# B&R Automation Studio project MVP_ACOPOStrak
Automation Studio 4.7.4.67 SP; technology packages: mapp 5.9.1, mappCockpit 5.9.0, mappMotion 5.9.2, mappView 5.9.1

## Configuration ACOPOStrak

CPU 5PC900.TS17-00, AutomationRuntime C4.72, Build 4.1.2, Safety 0.0, Vc V4.53.0

### IoMap.iom - 5PC900_TS17_00/IoMap.iom
```iecst
VAR_CONFIG
	::Safety:moduleOK AT %IX."epl_icn".ModuleOk;
	::Safety:resetNeeded AT %IX."epl_icn".resetNeeded;
	::Safety:resetSafety AT %QX."epl_icn".resetCommand;
	::Safety:safetyStarted AT %IX."epl_icn".safetyStarted;
	::Safety:safetyOK AT %IX."epl_icn".safetyOK;
END_VAR
```

## Configuration Safety

### Task classes (Cpu.sw)
```
Cyclic#4:
  Safety <- Safety.prg
  PB1 <- PB1.prg
  PP1 <- PP1.prg
  PP2 <- PP2.prg
  PB2 <- PB2.prg
  PP3 <- PP3.prg
  PB3 <- PB3.prg
  PP4 <- PP4.prg
  PP5 <- PP5.prg
Binaries: arsvcreg, udbdef, TCData, arflatprv, arcoal, mvLoader, FWRules, mCoWebSc, ashwd, ashwac, User, sysconf, asfw, arconfig, Role, iomap, Config
Libraries: DataObj, AsXml, standard, runtime, FileIO, astime, mpbase, SfDomVis, asiodiag, asieccon, aruser, brsystem, SfDomDrv, sys_lib, MpSfDomMgr, asusb, astcp
```

- Safety project (password-protected, skipped)

## Configuration Simulation

### Task classes (Cpu.sw)
```
Cyclic#1:
  Safety <- Safety.prg
  Receip_Han <- SequenceHandler.prg
  PB1 <- PB1.prg
  PP1 <- PP1.prg
  PP2 <- PP2.prg
  PB2 <- PB2.prg
  PP3 <- PP3.prg
  PB3 <- PB3.prg
  PP4 <- PP4.prg
  PP5 <- PP5.prg
  Vis <- Vis.prg
  StartMovem <- StartMovement.prg
DataObjects: McAcpSys
Binaries: TCData, udbdef, mvLoader, mCoWebSc, arsvcreg, McAcpDrv, Config_5, Config_4, AlarmCore, AlarmHist, Settings, ashwac, arconfig, asfw, TraceConfi, User, ashwd, iomap, Role, sysconf, Config_1, Config_3, Config_2, McAcpSim, McProfGen
Libraries: McAxis, McBase, McAcpTrak, brsystem, AsSem, sys_lib, runtime, operator, astime, AsIecCon, CoTrace, AsZip, FileIO, MpAlarmX, MpBase, MpAxis, McAcpAx, AsBrStr, AsIODiag, arflatprv, arcoal, powerlnk, dataobj, standard, MpSfDomMgr, SfDomDrv, SfDomVis, aruser, asusb, astcp
```

### Hardware
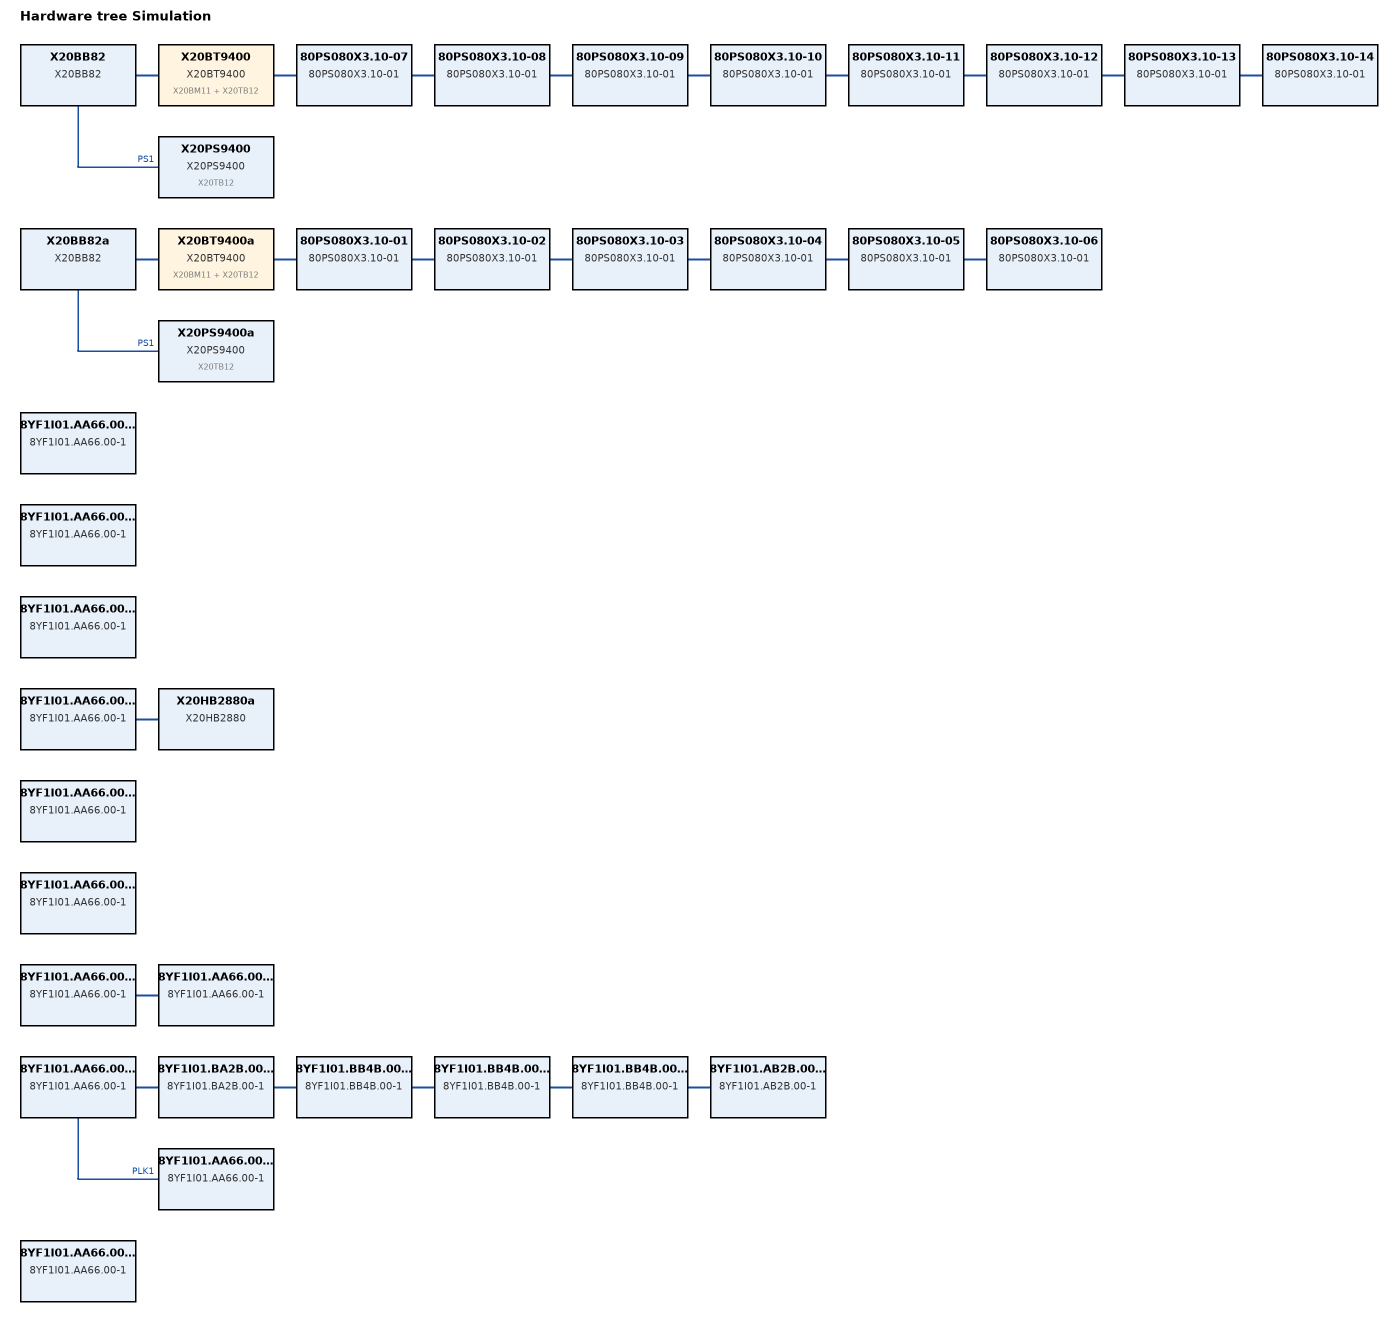
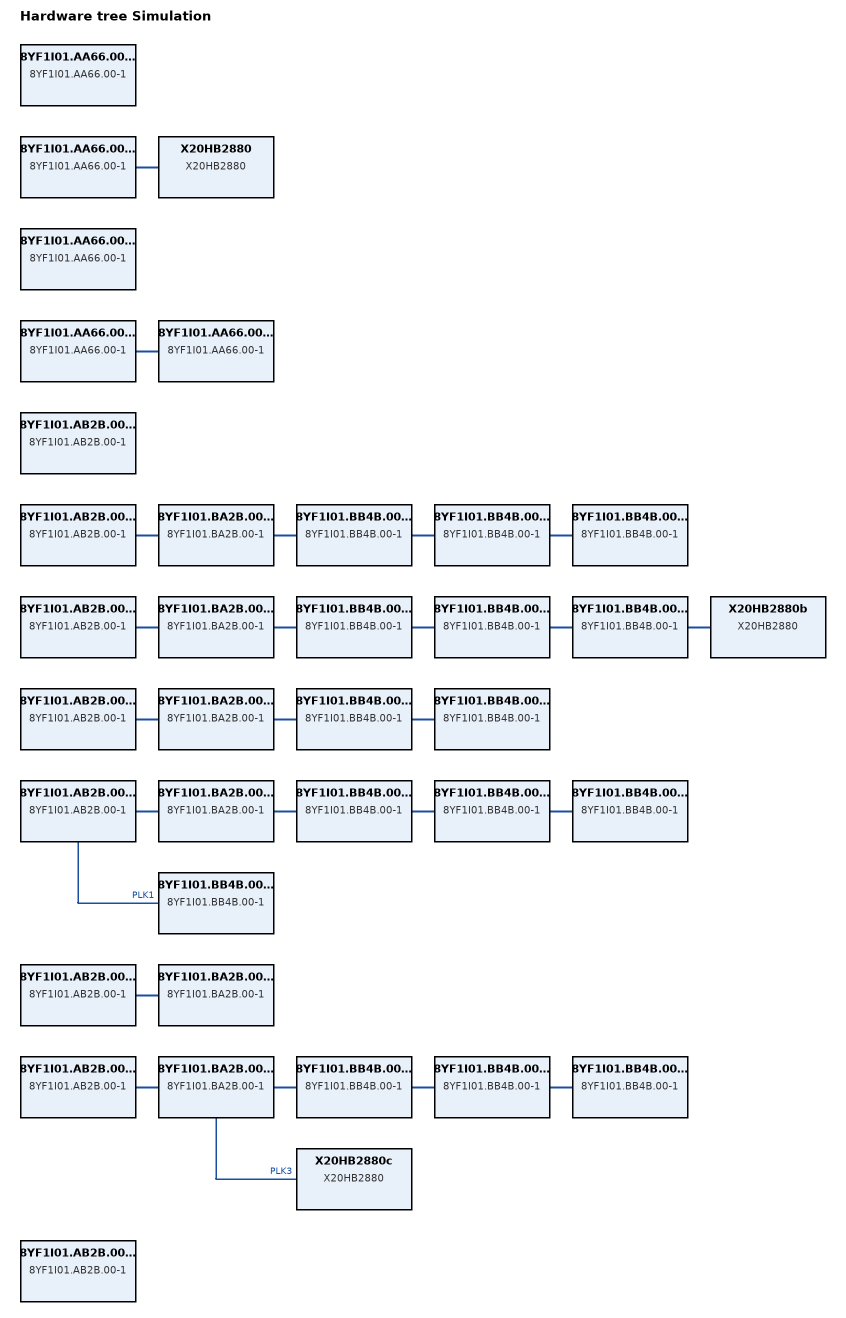
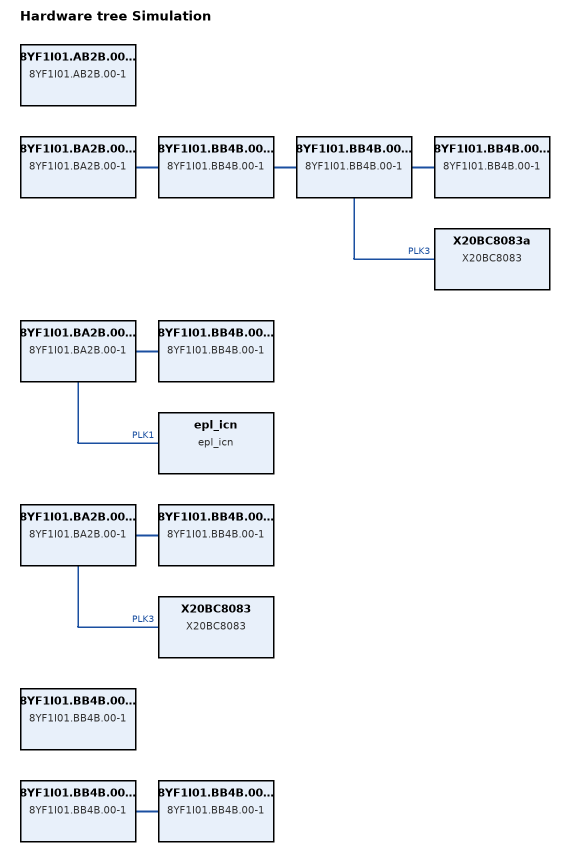
```
80PS080X3.10-01 : 80PS080X3.10-01 v1.3.0.0  [X2X1 -> X20BT9400a.X2X1 [Cable Type=X2XCable, Length=3, Version=1.0.0.2]]
  Supervision = off
  ParallelMode01 = on
  VoltageSet01 = 60
  ChopperEnable01 = on
80PS080X3.10-02 : 80PS080X3.10-01 v1.3.0.0  [X2X1 -> 80PS080X3.10-01.X2X2 [Cable Type=X2XCable, Length=1, Version=1.0.0.2]]
  Supervision = off
  ParallelMode01 = on
  VoltageSet01 = 60
  ChopperEnable01 = on
80PS080X3.10-03 : 80PS080X3.10-01 v1.3.0.0  [X2X1 -> 80PS080X3.10-02.X2X2 [Cable Type=X2XCable, Length=5, Version=1.0.0.2]]
  Supervision = off
  VoltageSet01 = 58
  ChopperEnable01 = on
80PS080X3.10-04 : 80PS080X3.10-01 v1.3.0.0  [X2X1 -> 80PS080X3.10-03.X2X2 [Cable Type=X2XCable, Length=1, Version=1.0.0.2]]
  Supervision = off
  VoltageSet01 = 58
  ChopperEnable01 = on
80PS080X3.10-05 : 80PS080X3.10-01 v1.3.0.0  [X2X1 -> 80PS080X3.10-04.X2X2 [Cable Type=X2XCable, Length=5, Version=1.0.0.2]]
  Supervision = off
  VoltageSet01 = 58
  ChopperEnable01 = on
80PS080X3.10-06 : 80PS080X3.10-01 v1.3.0.0  [X2X1 -> 80PS080X3.10-05.X2X2 [Cable Type=X2XCable, Length=1, Version=1.0.0.2]]
  Supervision = off
  VoltageSet01 = 58
  ChopperEnable01 = on
80PS080X3.10-07 : 80PS080X3.10-01 v1.3.0.0  [X2X1 -> X20BT9400.X2X1 [Cable Type=X2XCable, Length=5, Version=1.0.0.2]]
  Supervision = off
  VoltageSet01 = 58
  ChopperEnable01 = on
80PS080X3.10-08 : 80PS080X3.10-01 v1.3.0.0  [X2X1 -> 80PS080X3.10-07.X2X2 [Cable Type=X2XCable, Length=1, Version=1.0.0.2]]
  Supervision = off
  VoltageSet01 = 58
  ChopperEnable01 = on
80PS080X3.10-09 : 80PS080X3.10-01 v1.3.0.0  [X2X1 -> 80PS080X3.10-08.X2X2 [Cable Type=X2XCable, Length=1, Version=1.0.0.2]]
  Supervision = off
  VoltageSet01 = 58
  ChopperEnable01 = on
80PS080X3.10-10 : 80PS080X3.10-01 v1.3.0.0  [X2X1 -> 80PS080X3.10-09.X2X2 [Cable Type=X2XCable, Length=1, Version=1.0.0.2]]
  Supervision = off
  VoltageSet01 = 58
  ChopperEnable01 = on
80PS080X3.10-11 : 80PS080X3.10-01 v1.3.0.0  [X2X1 -> 80PS080X3.10-10.X2X2 [Cable Type=X2XCable, Length=3, Version=1.0.0.2]]
  Supervision = off
  VoltageSet01 = 58
  ChopperEnable01 = on
80PS080X3.10-12 : 80PS080X3.10-01 v1.3.0.0  [X2X1 -> 80PS080X3.10-11.X2X2 [Cable Type=X2XCable, Length=1, Version=1.0.0.2]]
  Supervision = off
  VoltageSet01 = 58
  ChopperEnable01 = on
80PS080X3.10-13 : 80PS080X3.10-01 v1.3.0.0  [X2X1 -> 80PS080X3.10-12.X2X2 [Cable Type=X2XCable, Length=1, Version=1.0.0.2]]
  Supervision = off
  VoltageSet01 = 58
  ChopperEnable01 = on
80PS080X3.10-14 : 80PS080X3.10-01 v1.3.0.0  [X2X1 -> 80PS080X3.10-13.X2X2 [Cable Type=X2XCable, Length=1, Version=1.0.0.2]]
  Supervision = off
  VoltageSet01 = 58
  ChopperEnable01 = on
8YF1I01.AA66.00-1_16 : 8YF1I01.AA66.00-1 v0.0.0.4  [PLK1 -> 8YF1I01.AA66.00-1_17.PLK2 (NodeNumber=16) [Cable Type=PowerlinkCable, Length=10, Version=1.0.0.2]]
  DriveConfiguration:
    McTypeID = LLMConfig
  DriveConfiguration/Segment:
    Shape = STRAIGHT660
    SegmentReference = SEG_1_16
    StopReaction = UseAssemblySetting
    SpeedFilter = UseAssemblySetting
8YF1I01.AA66.00-1_17 : 8YF1I01.AA66.00-1 v0.0.0.4  [PLK1 -> 8YF1I01.AA66.00-1_18.PLK2 (NodeNumber=17) [Cable Type=PowerlinkCable, Length=10, Version=1.0.0.2]; PLK2 -> 8YF1I01.AA66.00-1_16.PLK1 (NodeNumber=17) [Cable Type=PowerlinkCable, Length=10, Version=1.0.0.2]]
  DriveConfiguration:
    McTypeID = LLMConfig
  DriveConfiguration/Segment:
    Shape = STRAIGHT660
    SegmentReference = SEG_1_17
    StopReaction = UseAssemblySetting
    SpeedFilter = UseAssemblySetting
8YF1I01.AA66.00-1_18 : 8YF1I01.AA66.00-1 v0.0.0.4  [PLK1 -> 8YF1I01.AA66.00-1_19.PLK2 (NodeNumber=18) [Cable Type=PowerlinkCable, Length=10, Version=1.0.0.2]; PLK2 -> 8YF1I01.AA66.00-1_17.PLK1 (NodeNumber=18) [Cable Type=PowerlinkCable, Length=10, Version=1.0.0.2]]
  DriveConfiguration:
    McTypeID = LLMConfig
  DriveConfiguration/Segment:
    Shape = STRAIGHT660
    SegmentReference = SEG_1_18
    StopReaction = UseAssemblySetting
    SpeedFilter = UseAssemblySetting
8YF1I01.AA66.00-1_19 : 8YF1I01.AA66.00-1 v0.0.0.4  [PLK1 -> 8YF1I01.AA66.00-1_20.PLK2 (NodeNumber=19) [Cable Type=PowerlinkCable, Length=10, Version=1.0.0.2]; PLK2 -> 8YF1I01.AA66.00-1_18.PLK1 (NodeNumber=19) [Cable Type=PowerlinkCable, Length=10, Version=1.0.0.2]; PLK3 -> X20HB2880a.ETH1 (NodeNumber=19) [Cable Type=PowerlinkCable, Length=10, Version=1.0.0.2]]
  DriveConfiguration:
    McTypeID = LLMConfig
  DriveConfiguration/Segment:
    Shape = STRAIGHT660
    SegmentReference = SEG_1_19
    StopReaction = UseAssemblySetting
    SpeedFilter = UseAssemblySetting
8YF1I01.AA66.00-1_20 : 8YF1I01.AA66.00-1 v0.0.0.4  [PLK1 -> 8YF1I01.AA66.00-1_21.PLK2 (NodeNumber=20) [Cable Type=PowerlinkCable, Length=10, Version=1.0.0.2]; PLK2 -> 8YF1I01.AA66.00-1_19.PLK1 (NodeNumber=20) [Cable Type=PowerlinkCable, Length=10, Version=1.0.0.2]]
  DriveConfiguration:
    McTypeID = LLMConfig
  DriveConfiguration/Segment:
    Shape = STRAIGHT660
    SegmentReference = SEG_1_20
    StopReaction = UseAssemblySetting
    SpeedFilter = UseAssemblySetting
8YF1I01.AA66.00-1_21 : 8YF1I01.AA66.00-1 v0.0.0.4  [PLK1 -> 8YF1I01.AA66.00-1_22.PLK2 [Cable Type=PowerlinkCable, Length=10, Version=1.0.0.2]; PLK2 -> 8YF1I01.AA66.00-1_20.PLK1 [Cable Type=PowerlinkCable, Length=10, Version=1.0.0.2]]
  DriveConfiguration:
    McTypeID = LLMConfig
  DriveConfiguration/Segment:
    Shape = STRAIGHT660
    SegmentReference = SEG_1_21
    StopReaction = UseAssemblySetting
    SpeedFilter = UseAssemblySetting
8YF1I01.AA66.00-1_22 : 8YF1I01.AA66.00-1 v0.0.0.4  [PLK1 -> 8YF1I01.AA66.00-1_23.PLK2 [Cable Type=PowerlinkCable, Length=10, Version=1.0.0.2]; PLK2 -> 8YF1I01.AA66.00-1_21.PLK1 [Cable Type=PowerlinkCable, Length=10, Version=1.0.0.2]]
  DriveConfiguration:
    McTypeID = LLMConfig
  DriveConfiguration/Segment:
    Shape = STRAIGHT660
    SegmentReference = SEG_1_22
    StopReaction = UseAssemblySetting
    SpeedFilter = UseAssemblySetting
8YF1I01.AA66.00-1_23 : 8YF1I01.AA66.00-1 v0.0.0.4  [PLK2 -> 8YF1I01.AA66.00-1_22.PLK1 [Cable Type=PowerlinkCable, Length=10, Version=1.0.0.2]]
  DriveConfiguration:
    McTypeID = LLMConfig
  DriveConfiguration/Segment:
    Shape = STRAIGHT660
    SegmentReference = SEG_1_23
    StopReaction = UseAssemblySetting
    SpeedFilter = UseAssemblySetting
8YF1I01.AA66.00-1_29 : 8YF1I01.AA66.00-1 v0.0.0.4  [PLK1 -> 8YF1I01.AA66.00-1_30.PLK2 [Cable Type=PowerlinkCable, Length=10, Version=1.0.0.2]; PLK2 -> 8YF1I01.BA2B.00-1_28.PLK1 [Cable Type=PowerlinkCable, Length=10, Version=1.0.0.2]]
  DriveConfiguration:
    McTypeID = LLMConfig
  DriveConfiguration/Segment:
    Shape = STRAIGHT660
    SegmentReference = SEG_1_29
    StopReaction = UseAssemblySetting
    SpeedFilter = UseAssemblySetting
8YF1I01.AA66.00-1_30 : 8YF1I01.AA66.00-1 v0.0.0.4  [PLK2 -> 8YF1I01.AA66.00-1_29.PLK1 (NodeNumber=30) [Cable Type=PowerlinkCable, Length=10, Version=1.0.0.2]]
  DriveConfiguration:
    McTypeID = LLMConfig
  DriveConfiguration/Segment:
    Shape = STRAIGHT660
    SegmentReference = SEG_1_30
    StopReaction = UseAssemblySetting
    SpeedFilter = UseAssemblySetting
8YF1I01.AA66.00-1_31 : 8YF1I01.AA66.00-1 v0.0.0.4  [PLK1 -> 8YF1I01.AA66.00-1_32.PLK2 (NodeNumber=31) [Cable Type=PowerlinkCable, Length=10, Version=1.0.0.2]]
  DriveConfiguration:
    McTypeID = LLMConfig
  DriveConfiguration/Segment:
    Shape = STRAIGHT660
    SegmentReference = SEG_1_31
    StopReaction = UseAssemblySetting
    SpeedFilter = UseAssemblySetting
8YF1I01.AA66.00-1_32 : 8YF1I01.AA66.00-1 v0.0.0.4  [PLK1 -> 8YF1I01.AA66.00-1_33.PLK2 (NodeNumber=32) [Cable Type=PowerlinkCable, Length=10, Version=1.0.0.2]; PLK2 -> 8YF1I01.AA66.00-1_31.PLK1 (NodeNumber=32) [Cable Type=PowerlinkCable, Length=10, Version=1.0.0.2]]
  DriveConfiguration:
    McTypeID = LLMConfig
  DriveConfiguration/Segment:
    Shape = STRAIGHT660
    SegmentReference = SEG_1_32
    StopReaction = UseAssemblySetting
    SpeedFilter = UseAssemblySetting
8YF1I01.AA66.00-1_33 : 8YF1I01.AA66.00-1 v0.0.0.4  [PLK1 -> 8YF1I01.AA66.00-1_34.PLK2 (NodeNumber=33) [Cable Type=PowerlinkCable, Length=10, Version=1.0.0.2]; PLK2 -> 8YF1I01.AA66.00-1_32.PLK1 (NodeNumber=33) [Cable Type=PowerlinkCable, Length=10, Version=1.0.0.2]; PLK3 -> X20HB2880.ETH1 (NodeNumber=33) [Cable Type=PowerlinkCable, Length=10, Version=1.0.0.2]]
  DriveConfiguration:
    McTypeID = LLMConfig
  DriveConfiguration/Segment:
    Shape = STRAIGHT660
    SegmentReference = SEG_1_33
    StopReaction = UseAssemblySetting
    SpeedFilter = UseAssemblySetting
8YF1I01.AA66.00-1_34 : 8YF1I01.AA66.00-1 v0.0.0.4  [PLK1 -> 8YF1I01.AA66.00-1_35.PLK2 [Cable Type=PowerlinkCable, Length=10, Version=1.0.0.2]; PLK2 -> 8YF1I01.AA66.00-1_33.PLK1 [Cable Type=PowerlinkCable, Length=10, Version=1.0.0.2]]
  DriveConfiguration:
    McTypeID = LLMConfig
  DriveConfiguration/Segment:
    Shape = STRAIGHT660
    SegmentReference = SEG_1_34
    StopReaction = UseAssemblySetting
    SpeedFilter = UseAssemblySetting
8YF1I01.AA66.00-1_35 : 8YF1I01.AA66.00-1 v0.0.0.4  [PLK1 -> 8YF1I01.AA66.00-1_36.PLK2 [Cable Type=PowerlinkCable, Length=10, Version=1.0.0.2]; PLK2 -> 8YF1I01.AA66.00-1_34.PLK1 [Cable Type=PowerlinkCable, Length=10, Version=1.0.0.2]]
  DriveConfiguration:
    McTypeID = LLMConfig
  DriveConfiguration/Segment:
    Shape = STRAIGHT660
    SegmentReference = SEG_1_35
    StopReaction = UseAssemblySetting
    SpeedFilter = UseAssemblySetting
8YF1I01.AA66.00-1_36 : 8YF1I01.AA66.00-1 v0.0.0.4  [PLK2 -> 8YF1I01.AA66.00-1_35.PLK1 [Cable Type=PowerlinkCable, Length=10, Version=1.0.0.2]]
  DriveConfiguration:
    McTypeID = LLMConfig
  DriveConfiguration/Segment:
    Shape = STRAIGHT660
    SegmentReference = SEG_1_36
    StopReaction = UseAssemblySetting
    SpeedFilter = UseAssemblySetting
8YF1I01.AB2B.00-1_11 : 8YF1I01.AB2B.00-1 v0.0.0.4  [PLK1 -> 8YF1I01.BB4B.00-1_12.PLK2 (NodeNumber=11) [Cable Type=PowerlinkCable, Length=10, Version=1.0.0.2]]
  DriveConfiguration:
    McTypeID = LLMConfig
  DriveConfiguration/Segment:
    Shape = STRAIGHT105_TO_CIRCULAR
    SegmentReference = SEG_1_11
    StopReaction = UseAssemblySetting
    SpeedFilter = UseAssemblySetting
8YF1I01.AB2B.00-1_24 : 8YF1I01.AB2B.00-1 v0.0.0.4  [PLK1 -> 8YF1I01.BB4B.00-1_25.PLK2 (NodeNumber=24) [Cable Type=PowerlinkCable, Length=10, Version=1.0.0.2]]
  DriveConfiguration:
    McTypeID = LLMConfig
  DriveConfiguration/Segment:
    Shape = STRAIGHT105_TO_CIRCULAR
    SegmentReference = SEG_1_24
    StopReaction = UseAssemblySetting
    SpeedFilter = UseAssemblySetting
8YF1I01.AB2B.00-2_78 : 8YF1I01.AB2B.00-1 v0.0.0.4  [PLK1 -> 8YF1I01.BB4B.00-2_79.PLK2 (NodeNumber=78) [Cable Type=PowerlinkCable, Length=10, Version=1.0.0.2]; PLK2 -> 8YF1I01.BA2B.00-2_77.PLK1 (NodeNumber=78) [Cable Type=PowerlinkCable, Length=10, Version=1.0.0.2]]
  DriveConfiguration:
    McTypeID = LLMConfig
  DriveConfiguration/Segment:
    Shape = STRAIGHT105_TO_CIRCULAR
    SegmentReference = SEG_2_78
    StopReaction = UseAssemblySetting
    SpeedFilter = UseAssemblySetting
8YF1I01.AB2B.00-2_83 : 8YF1I01.AB2B.00-1 v0.0.0.4  [PLK2 -> 8YF1I01.BA2B.00-2_82.PLK1 [Cable Type=PowerlinkCable, Length=10, Version=1.0.0.2]]
  DriveConfiguration:
    McTypeID = LLMConfig
  DriveConfiguration/Segment:
    Shape = STRAIGHT105_TO_CIRCULAR
    SegmentReference = SEG_2_83
    StopReaction = UseAssemblySetting
    SpeedFilter = UseAssemblySetting
8YF1I01.AB2B.00-3_67 : 8YF1I01.AB2B.00-1 v0.0.0.4  [PLK1 -> 8YF1I01.BB4B.00-3_68.PLK2 (NodeNumber=67) [Cable Type=PowerlinkCable, Length=10, Version=1.0.0.2]; PLK2 -> 8YF1I01.BA2B.00-3_66.PLK1 (NodeNumber=67) [Cable Type=PowerlinkCable, Length=10, Version=1.0.0.2]]
  DriveConfiguration:
    McTypeID = LLMConfig
  DriveConfiguration/Segment:
    Shape = STRAIGHT105_TO_CIRCULAR
    SegmentReference = SEG_3_67
    StopReaction = UseAssemblySetting
    SpeedFilter = UseAssemblySetting
8YF1I01.AB2B.00-3_72 : 8YF1I01.AB2B.00-1 v0.0.0.4  [PLK1 -> 8YF1I01.BB4B.00-3_73.PLK2 [Cable Type=PowerlinkCable, Length=10, Version=1.0.0.2]; PLK2 -> 8YF1I01.BA2B.00-3_71.PLK1 [Cable Type=PowerlinkCable, Length=10, Version=1.0.0.2]]
  DriveConfiguration:
    McTypeID = LLMConfig
  DriveConfiguration/Segment:
    Shape = STRAIGHT105_TO_CIRCULAR
    SegmentReference = SEG_3_72
    StopReaction = UseAssemblySetting
    SpeedFilter = UseAssemblySetting
8YF1I01.AB2B.00-4_55 : 8YF1I01.AB2B.00-1 v0.0.0.4  [PLK1 -> 8YF1I01.BB4B.00-4_56.PLK2 (NodeNumber=55) [Cable Type=PowerlinkCable, Length=10, Version=1.0.0.2]; PLK2 -> 8YF1I01.BA2B.00-4_54.PLK1 (NodeNumber=55) [Cable Type=PowerlinkCable, Length=10, Version=1.0.0.2]]
  DriveConfiguration:
    McTypeID = LLMConfig
  DriveConfiguration/Segment:
    Shape = STRAIGHT105_TO_CIRCULAR
    SegmentReference = SEG_4_55
    StopReaction = UseAssemblySetting
    SpeedFilter = UseAssemblySetting
8YF1I01.AB2B.00-4_60 : 8YF1I01.AB2B.00-1 v0.0.0.4  [PLK1 -> 8YF1I01.BB4B.00-4_61.PLK2 [Cable Type=PowerlinkCable, Length=10, Version=1.0.0.2]; PLK2 -> 8YF1I01.BA2B.00-4_59.PLK1 [Cable Type=PowerlinkCable, Length=10, Version=1.0.0.2]]
  DriveConfiguration:
    McTypeID = LLMConfig
  DriveConfiguration/Segment:
    Shape = STRAIGHT105_TO_CIRCULAR
    SegmentReference = SEG_4_60
    StopReaction = UseAssemblySetting
    SpeedFilter = UseAssemblySetting
8YF1I01.AB2B.00-5_37 : 8YF1I01.AB2B.00-1 v0.0.0.4  [PLK1 -> 8YF1I01.BB4B.00-5_38.PLK2 (NodeNumber=37) [Cable Type=PowerlinkCable, Length=10, Version=1.0.0.2]; PLK3 -> X20HB2880.ETH2 (NodeNumber=37) [Cable Type=PowerlinkCable, Length=10, Version=1.0.0.2]]
  DriveConfiguration:
    McTypeID = LLMConfig
  DriveConfiguration/Segment:
    Shape = STRAIGHT105_TO_CIRCULAR
    SegmentReference = SEG_5_37
    StopReaction = UseAssemblySetting
    SpeedFilter = UseAssemblySetting
8YF1I01.AB2B.00-6_51 : 8YF1I01.AB2B.00-1 v0.0.0.4  [PLK1 -> 8YF1I01.BB4B.00-6_52.PLK2 (NodeNumber=51) [Cable Type=PowerlinkCable, Length=10, Version=1.0.0.2]]
  DriveConfiguration:
    McTypeID = LLMConfig
  DriveConfiguration/Segment:
    Shape = STRAIGHT105_TO_CIRCULAR
    SegmentReference = SEG_6_51
    StopReaction = UseAssemblySetting
    SpeedFilter = UseAssemblySetting
8YF1I01.BA2B.00-1_15 : 8YF1I01.BA2B.00-1 v0.0.0.4  [PLK2 -> 8YF1I01.BB4B.00-1_14.PLK1 [Cable Type=PowerlinkCable, Length=10, Version=1.0.0.2]]
  DriveConfiguration:
    McTypeID = LLMConfig
  DriveConfiguration/Segment:
    Shape = CIRCULAR_TO_STRAIGHT105
    SegmentReference = SEG_1_15
    StopReaction = UseAssemblySetting
    SpeedFilter = UseAssemblySetting
8YF1I01.BA2B.00-1_28 : 8YF1I01.BA2B.00-1 v0.0.0.4  [PLK1 -> 8YF1I01.AA66.00-1_29.PLK2 (NodeNumber=28) [Cable Type=PowerlinkCable, Length=10, Version=1.0.0.2]; PLK2 -> 8YF1I01.BB4B.00-1_27.PLK1 (NodeNumber=28) [Cable Type=PowerlinkCable, Length=10, Version=1.0.0.2]; PLK3 -> X20HB2880a.ETH2 (NodeNumber=28) [Cable Type=PowerlinkCable, Length=10, Version=1.0.0.2]]
  DriveConfiguration:
    McTypeID = LLMConfig
  DriveConfiguration/Segment:
    Shape = CIRCULAR_TO_STRAIGHT105
    SegmentReference = SEG_1_28
    StopReaction = UseAssemblySetting
    SpeedFilter = UseAssemblySetting
8YF1I01.BA2B.00-2_77 : 8YF1I01.BA2B.00-1 v0.0.0.4  [PLK1 -> 8YF1I01.AB2B.00-2_78.PLK2 (NodeNumber=77) [Cable Type=PowerlinkCable, Length=10, Version=1.0.0.2]; PLK2 -> 8YF1I01.BB4B.00-2_76.PLK1 (NodeNumber=77) [Cable Type=PowerlinkCable, Length=10, Version=1.0.0.2]]
  DriveConfiguration:
    McTypeID = LLMConfig
  DriveConfiguration/Segment:
    Shape = CIRCULAR_TO_STRAIGHT105
    SegmentReference = SEG_2_77
    StopReaction = UseAssemblySetting
    SpeedFilter = UseAssemblySetting
8YF1I01.BA2B.00-2_82 : 8YF1I01.BA2B.00-1 v0.0.0.4  [PLK1 -> 8YF1I01.AB2B.00-2_83.PLK2 [Cable Type=PowerlinkCable, Length=10, Version=1.0.0.2]; PLK2 -> 8YF1I01.BB4B.00-2_81.PLK1 [Cable Type=PowerlinkCable, Length=10, Version=1.0.0.2]]
  DriveConfiguration:
    McTypeID = LLMConfig
  DriveConfiguration/Segment:
    Shape = CIRCULAR_TO_STRAIGHT105
    SegmentReference = SEG_2_82
    StopReaction = UseAssemblySetting
    SpeedFilter = UseAssemblySetting
8YF1I01.BA2B.00-3_66 : 8YF1I01.BA2B.00-1 v0.0.0.4  [PLK1 -> 8YF1I01.AB2B.00-3_67.PLK2 (NodeNumber=66) [Cable Type=PowerlinkCable, Length=10, Version=1.0.0.2]; PLK2 -> 8YF1I01.BB4B.00-3_65.PLK1 (NodeNumber=66) [Cable Type=PowerlinkCable, Length=10, Version=1.0.0.2]]
  DriveConfiguration:
    McTypeID = LLMConfig
  DriveConfiguration/Segment:
    Shape = CIRCULAR_TO_STRAIGHT105
    SegmentReference = SEG_3_66
    StopReaction = UseAssemblySetting
    SpeedFilter = UseAssemblySetting
8YF1I01.BA2B.00-3_71 : 8YF1I01.BA2B.00-1 v0.0.0.4  [PLK1 -> 8YF1I01.AB2B.00-3_72.PLK2 [Cable Type=PowerlinkCable, Length=10, Version=1.0.0.2]; PLK2 -> 8YF1I01.BB4B.00-3_70.PLK1 [Cable Type=PowerlinkCable, Length=10, Version=1.0.0.2]]
  DriveConfiguration:
    McTypeID = LLMConfig
  DriveConfiguration/Segment:
    Shape = CIRCULAR_TO_STRAIGHT105
    SegmentReference = SEG_3_71
    StopReaction = UseAssemblySetting
    SpeedFilter = UseAssemblySetting
8YF1I01.BA2B.00-4_54 : 8YF1I01.BA2B.00-1 v0.0.0.4  [PLK1 -> 8YF1I01.AB2B.00-4_55.PLK2 (NodeNumber=54) [Cable Type=PowerlinkCable, Length=10, Version=1.0.0.2]]
  DriveConfiguration:
    McTypeID = LLMConfig
  DriveConfiguration/Segment:
    Shape = CIRCULAR_TO_STRAIGHT105
    SegmentReference = SEG_4_54
    StopReaction = UseAssemblySetting
    SpeedFilter = UseAssemblySetting
8YF1I01.BA2B.00-4_59 : 8YF1I01.BA2B.00-1 v0.0.0.4  [PLK1 -> 8YF1I01.AB2B.00-4_60.PLK2 (NodeNumber=59) [Cable Type=PowerlinkCable, Length=10, Version=1.0.0.2]; PLK2 -> 8YF1I01.BB4B.00-4_58.PLK1 (NodeNumber=59) [Cable Type=PowerlinkCable, Length=10, Version=1.0.0.2]; PLK3 -> X20HB2880c.ETH1 (NodeNumber=59) [Cable Type=PowerlinkCable, Length=10, Version=1.0.0.2]]
  DriveConfiguration:
    McTypeID = LLMConfig
  DriveConfiguration/Segment:
    Shape = CIRCULAR_TO_STRAIGHT105
    SegmentReference = SEG_4_59
    StopReaction = UseAssemblySetting
    SpeedFilter = UseAssemblySetting
8YF1I01.BA2B.00-5_39 : 8YF1I01.BA2B.00-1 v0.0.0.4  [PLK1 -> epl_icn.PLK1 [Cable Type=PowerlinkCable, Length=10, Version=1.0.0.2]; PLK2 -> 8YF1I01.BB4B.00-5_38.PLK1 [Cable Type=PowerlinkCable, Length=10, Version=1.0.0.2]]
  DriveConfiguration:
    McTypeID = LLMConfig
  DriveConfiguration/Segment:
    Shape = CIRCULAR_TO_STRAIGHT105
    SegmentReference = SEG_5_39
    StopReaction = UseAssemblySetting
    SpeedFilter = UseAssemblySetting
8YF1I01.BA2B.00-6_53 : 8YF1I01.BA2B.00-1 v0.0.0.4  [PLK2 -> 8YF1I01.BB4B.00-6_52.PLK1 (NodeNumber=53) [Cable Type=PowerlinkCable, Length=10, Version=1.0.0.2]; PLK3 -> X20BC8083.PLK2 (NodeNumber=53) [Cable Type=PowerlinkCable, Length=10, Version=1.0.0.2]]
  DriveConfiguration:
    McTypeID = LLMConfig
  DriveConfiguration/Segment:
    Shape = CIRCULAR_TO_STRAIGHT105
    SegmentReference = SEG_6_53
    StopReaction = UseAssemblySetting
    SpeedFilter = UseAssemblySetting
8YF1I01.BB4B.00-1_12 : 8YF1I01.BB4B.00-1 v0.0.0.4  [PLK1 -> 8YF1I01.BB4B.00-1_13.PLK2 (NodeNumber=12) [Cable Type=PowerlinkCable, Length=10, Version=1.0.0.2]; PLK2 -> 8YF1I01.AB2B.00-1_11.PLK1 (NodeNumber=12) [Cable Type=PowerlinkCable, Length=10, Version=1.0.0.2]]
  DriveConfiguration:
    McTypeID = LLMConfig
  DriveConfiguration/Segment:
    Shape = CIRCULAR
    SegmentReference = SEG_1_12
    StopReaction = UseAssemblySetting
    SpeedFilter = UseAssemblySetting
8YF1I01.BB4B.00-1_13 : 8YF1I01.BB4B.00-1 v0.0.0.4  [PLK1 -> 8YF1I01.BB4B.00-1_14.PLK2 (NodeNumber=13) [Cable Type=PowerlinkCable, Length=10, Version=1.0.0.2]; PLK2 -> 8YF1I01.BB4B.00-1_12.PLK1 (NodeNumber=13) [Cable Type=PowerlinkCable, Length=10, Version=1.0.0.2]; PLK3 -> X20BC8083a.PLK2 (NodeNumber=13) [Cable Type=PowerlinkCable, Length=10, Version=1.0.0.2]]
  DriveConfiguration:
    McTypeID = LLMConfig
  DriveConfiguration/Segment:
    Shape = CIRCULAR
    SegmentReference = SEG_1_13
    StopReaction = UseAssemblySetting
    SpeedFilter = UseAssemblySetting
8YF1I01.BB4B.00-1_14 : 8YF1I01.BB4B.00-1 v0.0.0.4  [PLK1 -> 8YF1I01.BA2B.00-1_15.PLK2 [Cable Type=PowerlinkCable, Length=10, Version=1.0.0.2]; PLK2 -> 8YF1I01.BB4B.00-1_13.PLK1 [Cable Type=PowerlinkCable, Length=10, Version=1.0.0.2]]
  DriveConfiguration:
    McTypeID = LLMConfig
  DriveConfiguration/Segment:
    Shape = CIRCULAR
    SegmentReference = SEG_1_14
    StopReaction = UseAssemblySetting
    SpeedFilter = UseAssemblySetting
8YF1I01.BB4B.00-1_25 : 8YF1I01.BB4B.00-1 v0.0.0.4  [PLK1 -> 8YF1I01.BB4B.00-1_26.PLK2 (NodeNumber=25) [Cable Type=PowerlinkCable, Length=10, Version=1.0.0.2]; PLK2 -> 8YF1I01.AB2B.00-1_24.PLK1 (NodeNumber=25) [Cable Type=PowerlinkCable, Length=10, Version=1.0.0.2]]
  DriveConfiguration:
    McTypeID = LLMConfig
  DriveConfiguration/Segment:
    Shape = CIRCULAR
    SegmentReference = SEG_1_25
    StopReaction = UseAssemblySetting
    SpeedFilter = UseAssemblySetting
8YF1I01.BB4B.00-1_26 : 8YF1I01.BB4B.00-1 v0.0.0.4  [PLK1 -> 8YF1I01.BB4B.00-1_27.PLK2 (NodeNumber=26) [Cable Type=PowerlinkCable, Length=10, Version=1.0.0.2]; PLK2 -> 8YF1I01.BB4B.00-1_25.PLK1 (NodeNumber=26) [Cable Type=PowerlinkCable, Length=10, Version=1.0.0.2]]
  DriveConfiguration:
    McTypeID = LLMConfig
  DriveConfiguration/Segment:
    Shape = CIRCULAR
    SegmentReference = SEG_1_26
    StopReaction = UseAssemblySetting
    SpeedFilter = UseAssemblySetting
8YF1I01.BB4B.00-1_27 : 8YF1I01.BB4B.00-1 v0.0.0.4  [PLK1 -> 8YF1I01.BA2B.00-1_28.PLK2 (NodeNumber=27) [Cable Type=PowerlinkCable, Length=10, Version=1.0.0.2]; PLK2 -> 8YF1I01.BB4B.00-1_26.PLK1 (NodeNumber=27) [Cable Type=PowerlinkCable, Length=10, Version=1.0.0.2]]
  DriveConfiguration:
    McTypeID = LLMConfig
  DriveConfiguration/Segment:
    Shape = CIRCULAR
    SegmentReference = SEG_1_27
    StopReaction = UseAssemblySetting
    SpeedFilter = UseAssemblySetting
8YF1I01.BB4B.00-2_74 : 8YF1I01.BB4B.00-1 v0.0.0.4  [PLK1 -> 8YF1I01.BB4B.00-2_75.PLK2 (NodeNumber=74) [Cable Type=PowerlinkCable, Length=10, Version=1.0.0.2]]
  DriveConfiguration:
    McTypeID = LLMConfig
  DriveConfiguration/Segment:
    Shape = CIRCULAR
    SegmentReference = SEG_2_74
    StopReaction = UseAssemblySetting
    SpeedFilter = UseAssemblySetting
8YF1I01.BB4B.00-2_75 : 8YF1I01.BB4B.00-1 v0.0.0.4  [PLK1 -> 8YF1I01.BB4B.00-2_76.PLK2 (NodeNumber=75) [Cable Type=PowerlinkCable, Length=10, Version=1.0.0.2]; PLK2 -> 8YF1I01.BB4B.00-2_74.PLK1 (NodeNumber=75) [Cable Type=PowerlinkCable, Length=10, Version=1.0.0.2]]
  DriveConfiguration:
    McTypeID = LLMConfig
  DriveConfiguration/Segment:
    Shape = CIRCULAR
    SegmentReference = SEG_2_75
    StopReaction = UseAssemblySetting
    SpeedFilter = UseAssemblySetting
8YF1I01.BB4B.00-2_76 : 8YF1I01.BB4B.00-1 v0.0.0.4  [PLK1 -> 8YF1I01.BA2B.00-2_77.PLK2 (NodeNumber=76) [Cable Type=PowerlinkCable, Length=10, Version=1.0.0.2]; PLK2 -> 8YF1I01.BB4B.00-2_75.PLK1 (NodeNumber=76) [Cable Type=PowerlinkCable, Length=10, Version=1.0.0.2]]
  DriveConfiguration:
    McTypeID = LLMConfig
  DriveConfiguration/Segment:
    Shape = CIRCULAR
    SegmentReference = SEG_2_76
    StopReaction = UseAssemblySetting
    SpeedFilter = UseAssemblySetting
8YF1I01.BB4B.00-2_79 : 8YF1I01.BB4B.00-1 v0.0.0.4  [PLK1 -> 8YF1I01.BB4B.00-2_80.PLK2 (NodeNumber=79) [Cable Type=PowerlinkCable, Length=10, Version=1.0.0.2]; PLK2 -> 8YF1I01.AB2B.00-2_78.PLK1 (NodeNumber=79) [Cable Type=PowerlinkCable, Length=10, Version=1.0.0.2]; PLK3 -> X20HB2880b.ETH1 (NodeNumber=79) [Cable Type=PowerlinkCable, Length=10, Version=1.0.0.2]]
  DriveConfiguration:
    McTypeID = LLMConfig
  DriveConfiguration/Segment:
    Shape = CIRCULAR
    SegmentReference = SEG_2_79
    StopReaction = UseAssemblySetting
    SpeedFilter = UseAssemblySetting
8YF1I01.BB4B.00-2_80 : 8YF1I01.BB4B.00-1 v0.0.0.4  [PLK1 -> 8YF1I01.BB4B.00-2_81.PLK2 [Cable Type=PowerlinkCable, Length=10, Version=1.0.0.2]; PLK2 -> 8YF1I01.BB4B.00-2_79.PLK1 [Cable Type=PowerlinkCable, Length=10, Version=1.0.0.2]]
  DriveConfiguration:
    McTypeID = LLMConfig
  DriveConfiguration/Segment:
    Shape = CIRCULAR
    SegmentReference = SEG_2_80
    StopReaction = UseAssemblySetting
    SpeedFilter = UseAssemblySetting
8YF1I01.BB4B.00-2_81 : 8YF1I01.BB4B.00-1 v0.0.0.4  [PLK1 -> 8YF1I01.BA2B.00-2_82.PLK2 [Cable Type=PowerlinkCable, Length=10, Version=1.0.0.2]; PLK2 -> 8YF1I01.BB4B.00-2_80.PLK1 [Cable Type=PowerlinkCable, Length=10, Version=1.0.0.2]]
  DriveConfiguration:
    McTypeID = LLMConfig
  DriveConfiguration/Segment:
    Shape = CIRCULAR
    SegmentReference = SEG_2_81
    StopReaction = UseAssemblySetting
    SpeedFilter = UseAssemblySetting
8YF1I01.BB4B.00-3_64 : 8YF1I01.BB4B.00-1 v0.0.0.4  [PLK1 -> 8YF1I01.BB4B.00-3_65.PLK2 (NodeNumber=64) [Cable Type=PowerlinkCable, Length=10, Version=1.0.0.2]]
  DriveConfiguration:
    McTypeID = LLMConfig
  DriveConfiguration/Segment:
    Shape = CIRCULAR
    SegmentReference = SEG_3_64
    StopReaction = UseAssemblySetting
    SpeedFilter = UseAssemblySetting
8YF1I01.BB4B.00-3_65 : 8YF1I01.BB4B.00-1 v0.0.0.4  [PLK1 -> 8YF1I01.BA2B.00-3_66.PLK2 (NodeNumber=65) [Cable Type=PowerlinkCable, Length=10, Version=1.0.0.2]; PLK2 -> 8YF1I01.BB4B.00-3_64.PLK1 (NodeNumber=65) [Cable Type=PowerlinkCable, Length=10, Version=1.0.0.2]]
  DriveConfiguration:
    McTypeID = LLMConfig
  DriveConfiguration/Segment:
    Shape = CIRCULAR
    SegmentReference = SEG_3_65
    StopReaction = UseAssemblySetting
    SpeedFilter = UseAssemblySetting
8YF1I01.BB4B.00-3_68 : 8YF1I01.BB4B.00-1 v0.0.0.4  [PLK1 -> 8YF1I01.BB4B.00-3_69.PLK2 (NodeNumber=68) [Cable Type=PowerlinkCable, Length=10, Version=1.0.0.2]; PLK2 -> 8YF1I01.AB2B.00-3_67.PLK1 (NodeNumber=68) [Cable Type=PowerlinkCable, Length=10, Version=1.0.0.2]]
  DriveConfiguration:
    McTypeID = LLMConfig
  DriveConfiguration/Segment:
    Shape = CIRCULAR
    SegmentReference = SEG_3_68
    StopReaction = UseAssemblySetting
    SpeedFilter = UseAssemblySetting
8YF1I01.BB4B.00-3_69 : 8YF1I01.BB4B.00-1 v0.0.0.4  [PLK1 -> 8YF1I01.BB4B.00-3_70.PLK2 (NodeNumber=69) [Cable Type=PowerlinkCable, Length=10, Version=1.0.0.2]; PLK2 -> 8YF1I01.BB4B.00-3_68.PLK1 (NodeNumber=69) [Cable Type=PowerlinkCable, Length=10, Version=1.0.0.2]; PLK3 -> X20HB2880c.ETH2 (NodeNumber=69) [Cable Type=PowerlinkCable, Length=10, Version=1.0.0.2]]
  DriveConfiguration:
    McTypeID = LLMConfig
  DriveConfiguration/Segment:
    Shape = CIRCULAR
    SegmentReference = SEG_3_69
    StopReaction = UseAssemblySetting
    SpeedFilter = UseAssemblySetting
8YF1I01.BB4B.00-3_70 : 8YF1I01.BB4B.00-1 v0.0.0.4  [PLK1 -> 8YF1I01.BA2B.00-3_71.PLK2 [Cable Type=PowerlinkCable, Length=10, Version=1.0.0.2]; PLK2 -> 8YF1I01.BB4B.00-3_69.PLK1 [Cable Type=PowerlinkCable, Length=10, Version=1.0.0.2]]
  DriveConfiguration:
    McTypeID = LLMConfig
  DriveConfiguration/Segment:
    Shape = CIRCULAR
    SegmentReference = SEG_3_70
    StopReaction = UseAssemblySetting
    SpeedFilter = UseAssemblySetting
8YF1I01.BB4B.00-3_73 : 8YF1I01.BB4B.00-1 v0.0.0.4  [PLK2 -> 8YF1I01.AB2B.00-3_72.PLK1 [Cable Type=PowerlinkCable, Length=10, Version=1.0.0.2]]
  DriveConfiguration:
    McTypeID = LLMConfig
  DriveConfiguration/Segment:
    Shape = CIRCULAR
    SegmentReference = SEG_3_73
    StopReaction = UseAssemblySetting
    SpeedFilter = UseAssemblySetting
8YF1I01.BB4B.00-4_56 : 8YF1I01.BB4B.00-1 v0.0.0.4  [PLK1 -> 8YF1I01.BB4B.00-4_57.PLK2 (NodeNumber=56) [Cable Type=PowerlinkCable, Length=10, Version=1.0.0.2]; PLK2 -> 8YF1I01.AB2B.00-4_55.PLK1 (NodeNumber=56) [Cable Type=PowerlinkCable, Length=10, Version=1.0.0.2]]
  DriveConfiguration:
    McTypeID = LLMConfig
  DriveConfiguration/Segment:
    Shape = CIRCULAR
    SegmentReference = SEG_4_56
    StopReaction = UseAssemblySetting
    SpeedFilter = UseAssemblySetting
8YF1I01.BB4B.00-4_57 : 8YF1I01.BB4B.00-1 v0.0.0.4  [PLK1 -> 8YF1I01.BB4B.00-4_58.PLK2 (NodeNumber=57) [Cable Type=PowerlinkCable, Length=10, Version=1.0.0.2]; PLK2 -> 8YF1I01.BB4B.00-4_56.PLK1 (NodeNumber=57) [Cable Type=PowerlinkCable, Length=10, Version=1.0.0.2]]
  DriveConfiguration:
    McTypeID = LLMConfig
  DriveConfiguration/Segment:
    Shape = CIRCULAR
    SegmentReference = SEG_4_57
    StopReaction = UseAssemblySetting
    SpeedFilter = UseAssemblySetting
8YF1I01.BB4B.00-4_58 : 8YF1I01.BB4B.00-1 v0.0.0.4  [PLK1 -> 8YF1I01.BA2B.00-4_59.PLK2 (NodeNumber=58) [Cable Type=PowerlinkCable, Length=10, Version=1.0.0.2]; PLK2 -> 8YF1I01.BB4B.00-4_57.PLK1 (NodeNumber=58) [Cable Type=PowerlinkCable, Length=10, Version=1.0.0.2]]
  DriveConfiguration:
    McTypeID = LLMConfig
  DriveConfiguration/Segment:
    Shape = CIRCULAR
    SegmentReference = SEG_4_58
    StopReaction = UseAssemblySetting
    SpeedFilter = UseAssemblySetting
8YF1I01.BB4B.00-4_61 : 8YF1I01.BB4B.00-1 v0.0.0.4  [PLK1 -> 8YF1I01.BB4B.00-4_62.PLK2 [Cable Type=PowerlinkCable, Length=10, Version=1.0.0.2]; PLK2 -> 8YF1I01.AB2B.00-4_60.PLK1 [Cable Type=PowerlinkCable, Length=10, Version=1.0.0.2]]
  DriveConfiguration:
    McTypeID = LLMConfig
  DriveConfiguration/Segment:
    Shape = CIRCULAR
    SegmentReference = SEG_4_61
    StopReaction = UseAssemblySetting
    SpeedFilter = UseAssemblySetting
8YF1I01.BB4B.00-4_62 : 8YF1I01.BB4B.00-1 v0.0.0.4  [PLK1 -> 8YF1I01.BB4B.00-4_63.PLK2 (NodeNumber=62) [Cable Type=PowerlinkCable, Length=10, Version=1.0.0.2]; PLK2 -> 8YF1I01.BB4B.00-4_61.PLK1 (NodeNumber=62) [Cable Type=PowerlinkCable, Length=10, Version=1.0.0.2]]
  DriveConfiguration:
    McTypeID = LLMConfig
  DriveConfiguration/Segment:
    Shape = CIRCULAR
    SegmentReference = SEG_4_62
    StopReaction = UseAssemblySetting
    SpeedFilter = UseAssemblySetting
8YF1I01.BB4B.00-4_63 : 8YF1I01.BB4B.00-1 v0.0.0.4  [PLK2 -> 8YF1I01.BB4B.00-4_62.PLK1 [Cable Type=PowerlinkCable, Length=10, Version=1.0.0.2]]
  DriveConfiguration:
    McTypeID = LLMConfig
  DriveConfiguration/Segment:
    Shape = CIRCULAR
    SegmentReference = SEG_4_63
    StopReaction = UseAssemblySetting
    SpeedFilter = UseAssemblySetting
8YF1I01.BB4B.00-5_38 : 8YF1I01.BB4B.00-1 v0.0.0.4  [PLK1 -> 8YF1I01.BA2B.00-5_39.PLK2 [Cable Type=PowerlinkCable, Length=10, Version=1.0.0.2]; PLK2 -> 8YF1I01.AB2B.00-5_37.PLK1 [Cable Type=PowerlinkCable, Length=10, Version=1.0.0.2]]
  DriveConfiguration:
    McTypeID = LLMConfig
  DriveConfiguration/Segment:
    Shape = CIRCULAR
    SegmentReference = SEG_5_38
    StopReaction = UseAssemblySetting
    SpeedFilter = UseAssemblySetting
8YF1I01.BB4B.00-6_52 : 8YF1I01.BB4B.00-1 v0.0.0.4  [PLK1 -> 8YF1I01.BA2B.00-6_53.PLK2 (NodeNumber=52) [Cable Type=PowerlinkCable, Length=10, Version=1.0.0.2]; PLK2 -> 8YF1I01.AB2B.00-6_51.PLK1 (NodeNumber=52) [Cable Type=PowerlinkCable, Length=10, Version=1.0.0.2]]
  DriveConfiguration:
    McTypeID = LLMConfig
  DriveConfiguration/Segment:
    Shape = CIRCULAR
    SegmentReference = SEG_6_52
    StopReaction = UseAssemblySetting
    SpeedFilter = UseAssemblySetting
X20BB82 : X20BB82 v1.0.2.0
  Connector IF1:
    CycleTime = 10000
    BusLength = 50
    Stations = 32
    AsyncPayload = 96
X20BB82a : X20BB82 v1.0.2.0
  Connector IF1:
    CycleTime = 10000
    BusLength = 50
    Stations = 32
    AsyncPayload = 96
X20BC8083 : X20BC8083 v2.10.0.0  [PLK1 -> 5LS182.6-2.IF1 (NodeNumber=50) [Cable Type=PowerlinkCable, Length=10, Version=1.0.0.2]; PLK2 -> 8YF1I01.BA2B.00-6_53.PLK3 (NodeNumber=50) [Cable Type=PowerlinkCable, Length=10, Version=1.0.0.2]; SL -> X20BB82.SL1]
  Supervision = off
X20BC8083a : X20BC8083 v2.10.0.0  [PLK1 -> 5LS182.6-2.PLK2 (NodeNumber=10) [Cable Type=PowerlinkCable, Length=10, Version=1.0.0.2]; PLK2 -> 8YF1I01.BB4B.00-1_13.PLK3 (NodeNumber=10) [Cable Type=PowerlinkCable, Length=10, Version=1.0.0.2]; SL -> X20BB82a.SL1]
  Supervision = off
X20BM11 : X20BM11 v1.0.0.1  [X2X1 -> X20BB82.IF1]
X20BM11a : X20BM11 v1.0.0.1  [X2X1 -> X20BB82a.IF1]
X20BT9400 : X20BT9400 v1.1.0.0  [SS1 -> X20TB12b.SS; SL -> X20BM11.SL1]
  Supervision = off
  PowerInfo = on
X20BT9400a : X20BT9400 v1.1.0.0  [SS1 -> X20TB12c.SS; SL -> X20BM11a.SL1]
  Supervision = off
  PowerInfo = on
X20HB2880 : X20HB2880 v1.1.0.0  [ETH1 -> 8YF1I01.AA66.00-1_33.PLK3 [Cable Type=PowerlinkCable, Length=10, Version=1.0.0.2]; ETH2 -> 8YF1I01.AB2B.00-5_37.PLK3 [Cable Type=PowerlinkCable, Length=10, Version=1.0.0.2]; SS -> X20BB82a.SS2]
X20HB2880a : X20HB2880 v1.1.0.0  [ETH1 -> 8YF1I01.AA66.00-1_19.PLK3 [Cable Type=PowerlinkCable, Length=10, Version=1.0.0.2]; ETH2 -> 8YF1I01.BA2B.00-1_28.PLK3 [Cable Type=PowerlinkCable, Length=10, Version=1.0.0.2]; SS -> X20BB82a.SS1]
X20HB2880b : X20HB2880 v1.1.0.0  [ETH1 -> 8YF1I01.BB4B.00-2_79.PLK3 [Cable Type=PowerlinkCable, Length=10, Version=1.0.0.2]; SS -> X20BB82.SS2]
X20HB2880c : X20HB2880 v1.1.0.0  [ETH1 -> 8YF1I01.BA2B.00-4_59.PLK3 [Cable Type=PowerlinkCable, Length=10, Version=1.0.0.2]; ETH2 -> 8YF1I01.BB4B.00-3_69.PLK3 [Cable Type=PowerlinkCable, Length=10, Version=1.0.0.2]; SS -> X20BB82.SS1]
X20PS9400 : X20PS9400 v1.3.0.0  [SS1 -> X20TB12.SS; PS -> X20BB82.PS1]
  Supervision = off
  PowerInfo = on
X20PS9400a : X20PS9400 v1.3.0.0  [SS1 -> X20TB12a.SS; PS -> X20BB82a.PS1]
  Supervision = off
  PowerInfo = on
X20TB12 : X20TB12 v1.0.0.0
X20TB12a : X20TB12 v1.0.0.0
X20TB12b : X20TB12 v1.0.0.0
X20TB12c : X20TB12 v1.0.0.0
epl_icn : epl_icn v1.3.2.0  [PLK1 -> 8YF1I01.BA2B.00-5_39.PLK1 (NodeNumber=200) [Cable Type=PowerlinkCable, Length=10, Version=1.0.0.2]]
  RefConfiguration = Safety
  RefInterface = X20CP0484.IF3
```

### Config_1.assembly - 5PC900_TS17_00/mappMotion/Config_1.assembly
```
Element gAssembly_1 (Type=assembly)
  Tracks:
    TrackSeparation = 0.030
    Track[1]:
      Segments:
        SegmentRef[1] = ::SEG_1_11
        SegmentRef[2] = ::SEG_1_12
        SegmentRef[3] = ::SEG_1_13
        SegmentRef[4] = ::SEG_1_14
        SegmentRef[5] = ::SEG_1_15
        SegmentRef[6] = ::SEG_1_16
        SegmentRef[7] = ::SEG_1_17
        SegmentRef[8] = ::SEG_1_18
        SegmentRef[9] = ::SEG_1_19
        SegmentRef[10] = ::SEG_1_20
        SegmentRef[11] = ::SEG_1_21
        SegmentRef[12] = ::SEG_1_22
        SegmentRef[13] = ::SEG_1_23
        SegmentRef[14] = ::SEG_1_24
        SegmentRef[15] = ::SEG_1_25
        SegmentRef[16] = ::SEG_1_26
        SegmentRef[17] = ::SEG_1_27
        SegmentRef[18] = ::SEG_1_28
        SegmentRef[19] = ::SEG_1_29
        SegmentRef[20] = ::SEG_1_30
        SegmentRef[21] = ::SEG_1_31
        SegmentRef[22] = ::SEG_1_32
        SegmentRef[23] = ::SEG_1_33
        SegmentRef[24] = ::SEG_1_34
        SegmentRef[25] = ::SEG_1_35
        SegmentRef[26] = ::SEG_1_36
      Position = Absolute
        SegmentRef = ::SEG_1_21
        SegmentCountDirection = RightToLeft
        Translation:
          X = 0.0
          Y = 0.0
          Z = 0.0
        Orientation:
          Angle1 = 0.0
          Angle2 = 0.0
          Angle3 = 0
    Track[2]:
      Segments:
        SegmentRef[1] = ::SEG_2_74
        SegmentRef[2] = ::SEG_2_75
        SegmentRef[3] = ::SEG_2_76
        SegmentRef[4] = ::SEG_2_77
        SegmentRef[5] = ::SEG_2_78
        SegmentRef[6] = ::SEG_2_79
        SegmentRef[7] = ::SEG_2_80
        SegmentRef[8] = ::SEG_2_81
        SegmentRef[9] = ::SEG_2_82
        SegmentRef[10] = ::SEG_2_83
      Position = RelativeToOne
        TrackSegmentPosition:
          SegmentRef = ::SEG_2_77
          PositionRelativeTo = FromEnd
        Base:
          SegmentRef = ::SEG_1_29
          Position = 0.321
    Track[3]:
      Segments:
        SegmentRef[1] = ::SEG_3_64
        SegmentRef[2] = ::SEG_3_65
        SegmentRef[3] = ::SEG_3_66
        SegmentRef[4] = ::SEG_3_67
        SegmentRef[5] = ::SEG_3_68
        SegmentRef[6] = ::SEG_3_69
        SegmentRef[7] = ::SEG_3_70
        SegmentRef[8] = ::SEG_3_71
        SegmentRef[9] = ::SEG_3_72
        SegmentRef[10] = ::SEG_3_73
      Position = RelativeToOne
        TrackSegmentPosition:
          SegmentRef = ::SEG_3_66
          PositionRelativeTo = FromEnd
        Base:
          SegmentRef = ::SEG_1_34
          Position = 0.33
    Track[4]:
      Segments:
        SegmentRef[1] = ::SEG_4_54
        SegmentRef[2] = ::SEG_4_55
        SegmentRef[3] = ::SEG_4_56
        SegmentRef[4] = ::SEG_4_57
        SegmentRef[5] = ::SEG_4_58
        SegmentRef[6] = ::SEG_4_59
        SegmentRef[7] = ::SEG_4_60
        SegmentRef[8] = ::SEG_4_61
        SegmentRef[9] = ::SEG_4_62
        SegmentRef[10] = ::SEG_4_63
      Position = RelativeToOne
        TrackSegmentPosition:
          SegmentRef = ::SEG_4_59
          PositionRelativeTo = FromEnd
        Base:
          SegmentRef = ::SEG_1_19
          Position = 0.33
    Track[5]:
      Segments:
        SegmentRef[1] = ::SEG_5_37
        SegmentRef[2] = ::SEG_5_38
        SegmentRef[3] = ::SEG_5_39
      Position = RelativeToOne
        TrackSegmentPosition:
          SegmentRef = ::SEG_5_39
          PositionRelativeTo = FromEnd
        Base:
          SegmentRef = ::SEG_1_11
    Track[6]:
      Segments:
        SegmentRef[1] = ::SEG_6_51
        SegmentRef[2] = ::SEG_6_52
        SegmentRef[3] = ::SEG_6_53
      Position = RelativeToOne
        TrackSegmentPosition:
          SegmentRef = ::SEG_6_51
        Base:
          SegmentRef = ::SEG_1_15
          PositionRelativeTo = FromEnd
  CommonSegmentSettings:
    SegmentSimulationOnPLC = Off
    StopReaction = InductionHalt
    SpeedFilter = Lowpass
      FilterTime = 0.0004
    ControllerParameters:
      DefaultParameter:
        Controller:
          Position:
            ProportionalGain = 150.0
          Speed:
            ProportionalGain = 80.0
            IntegrationTime = 0.0
          FeedForward:
            TotalMass = 0.0
            ForcePositive = 0.0
            ForceNegative = 0.0
            SpeedForceFactor = 0.0
            ForceLoad = 0.0
        MovementErrorLimits:
          PositionError = 1.0
          VelocityError = 10.0
      AdditionalParameterSets = NotUsed
  Shuttles:
    MaxShuttleCount = 40
    ShuttleStereotypes:
      ShuttleStRef[1] = ShuttleStereotype_1
    MagnetPlateConfigurations:
      ShuttleType[1] = 8F1SA.100.xxxxxx-x
    CollisionAvoidance:
      Strategy = Constant
      MaximumModelDimensions:
        Length:
          ExtentToFront = 0.065
          ExtentToBack = 0.065
        Width:
          Width = 0.240
  AssemblyFeatures:
    AssemblyFeatureRef[1] = AssemblyFeature_2
  Visualization:
    MonitoringPv = ::gShuttleMon
    ProcessingTaskClass = 1
```

### Config_2.shuttlestereotype - 5PC900_TS17_00/mappMotion/Config_2.shuttlestereotype
```
Element ShuttleStereotype_1 (Type=shuttlestereotype)
  MeasurementUnit = 5067858
  MeasurementResolution = 0.00001
  MovementLimits = Internal
    VelocityIsReadOnly = 0
    Velocity:
      Velocity = 5
    AccelerationIsReadOnly = 0
    Acceleration:
      Acceleration = 50
    DecelerationIsReadOnly = 0
    Deceleration:
      Deceleration = 50
  JerkFilter = Used
    JerkTime = 0.02
  UserData:
    Size = 12
  CollisionAvoidance:
    InitialModelDimensions = UseExplicitValues
      Length:
        ExtentToFront = 0.040
        ExtentToBack = 0.040
      Width:
        Width = 0.080
```

### Config_3.sector - 5PC900_TS17_00/mappMotion/Config_3.sector
```
Element SectorTrack1 (Type=sector)
  Type = Composed
    StartSegment:
      SegmentRef = ::SEG_1_11
    IntermediateSegments:
      SegmentRef[1] = ::SEG_1_12
      SegmentRef[2] = ::SEG_1_13
      SegmentRef[3] = ::SEG_1_14
      SegmentRef[4] = ::SEG_1_15
      SegmentRef[5] = ::SEG_1_16
      SegmentRef[6] = ::SEG_1_17
      SegmentRef[7] = ::SEG_1_18
      SegmentRef[8] = ::SEG_1_19
      SegmentRef[9] = ::SEG_1_20
      SegmentRef[10] = ::SEG_1_21
      SegmentRef[11] = ::SEG_1_22
      SegmentRef[12] = ::SEG_1_23
      SegmentRef[13] = ::SEG_1_24
      SegmentRef[14] = ::SEG_1_25
      SegmentRef[15] = ::SEG_1_26
      SegmentRef[16] = ::SEG_1_27
      SegmentRef[17] = ::SEG_1_28
      SegmentRef[18] = ::SEG_1_29
      SegmentRef[19] = ::SEG_1_30
      SegmentRef[20] = ::SEG_1_31
      SegmentRef[21] = ::SEG_1_32
      SegmentRef[22] = ::SEG_1_33
      SegmentRef[23] = ::SEG_1_34
      SegmentRef[24] = ::SEG_1_35
    EndSegment:
      SegmentRef = ::SEG_1_36
      PositionRelativeTo = FromEnd
Element SectorTrack2 (Type=sector)
  Type = Composed
    StartSegment:
      SegmentRef = ::SEG_2_74
    IntermediateSegments:
      SegmentRef[1] = ::SEG_2_75
      SegmentRef[2] = ::SEG_2_76
      SegmentRef[3] = ::SEG_2_77
      SegmentRef[4] = ::SEG_2_78
      SegmentRef[5] = ::SEG_2_79
      SegmentRef[6] = ::SEG_2_80
      SegmentRef[7] = ::SEG_2_81
      SegmentRef[8] = ::SEG_2_82
    EndSegment:
      SegmentRef = ::SEG_2_83
      PositionRelativeTo = FromEnd
Element SectorTrack3 (Type=sector)
  Type = Composed
    StartSegment:
      SegmentRef = ::SEG_3_64
    IntermediateSegments:
      SegmentRef[1] = ::SEG_3_65
      SegmentRef[2] = ::SEG_3_66
      SegmentRef[3] = ::SEG_3_67
      SegmentRef[4] = ::SEG_3_68
      SegmentRef[5] = ::SEG_3_69
      SegmentRef[6] = ::SEG_3_70
      SegmentRef[7] = ::SEG_3_71
      SegmentRef[8] = ::SEG_3_72
    EndSegment:
      SegmentRef = ::SEG_3_73
      PositionRelativeTo = FromEnd
Element SectorTrack4 (Type=sector)
  Type = Composed
    StartSegment:
      SegmentRef = ::SEG_4_54
    IntermediateSegments:
      SegmentRef[1] = ::SEG_4_55
      SegmentRef[2] = ::SEG_4_56
      SegmentRef[3] = ::SEG_4_57
      SegmentRef[4] = ::SEG_4_58
      SegmentRef[5] = ::SEG_4_59
      SegmentRef[6] = ::SEG_4_60
      SegmentRef[7] = ::SEG_4_61
      SegmentRef[8] = ::SEG_4_62
    EndSegment:
      SegmentRef = ::SEG_4_63
      PositionRelativeTo = FromEnd
Element SectorTrack5 (Type=sector)
  Type = Composed
    StartSegment:
      SegmentRef = ::SEG_5_37
    IntermediateSegments:
      SegmentRef[1] = ::SEG_5_38
    EndSegment:
      SegmentRef = ::SEG_5_39
      PositionRelativeTo = FromEnd
Element SectorTrack6 (Type=sector)
  Type = Composed
    StartSegment:
      SegmentRef = ::SEG_6_53
      PositionRelativeTo = FromEnd
    IntermediateSegments:
      SegmentRef[1] = ::SEG_6_52
    EndSegment:
      SegmentRef = ::SEG_6_51
Element SubSector1_1 (Type=sector)
  Type = Composed
    StartSegment:
      SegmentRef = ::SEG_1_14
    IntermediateSegments:
      SegmentRef[1] = ::SEG_1_15
    EndSegment:
      SegmentRef = ::SEG_1_16
      PositionRelativeTo = FromEnd
Element SubSector1_2 (Type=sector)
  Type = Composed
    StartSegment:
      SegmentRef = ::SEG_1_27
    EndSegment:
      SegmentRef = ::SEG_1_28
      PositionRelativeTo = FromEnd
Element SubSector1_3 (Type=sector)
  Type = Composed
    StartSegment:
      SegmentRef = ::SEG_1_33
    EndSegment:
      SegmentRef = ::SEG_1_34
      PositionRelativeTo = FromEnd
Element SubSector1_4 (Type=sector)
  Type = Composed
    StartSegment:
      SegmentRef = ::SEG_1_36
    EndSegment:
      SegmentRef = ::SEG_1_11
      PositionRelativeTo = FromEnd
Element SubSector2_1 (Type=sector)
  Type = Composed
    StartSegment:
      SegmentRef = ::SEG_2_82
    EndSegment:
      SegmentRef = ::SEG_2_83
      PositionRelativeTo = FromEnd
Element SubSector3_1 (Type=sector)
  Type = Composed
    StartSegment:
      SegmentRef = ::SEG_3_71
    EndSegment:
      SegmentRef = ::SEG_3_72
      PositionRelativeTo = FromEnd
```

### Config_4.processpointlist - 5PC900_TS17_00/mappMotion/Config_4.processpointlist
```
Element ProcessPointList_Sector (Type=processpointlist)
  ProcessPoint[0]:
    Name = PB1
    SectorRef = SubSector1_1
    Position = 0.1
    TriggerEventBufferSize = 10
    BarrierFunctionality = On
  ProcessPoint[1]:
    Name = PP1
    SectorRef = SubSector1_1
    Position = 0.3
    TriggerEventBufferSize = 10
    BarrierFunctionality = On
  ProcessPoint[2]:
    Name = PP2
    SectorRef = SubSector1_2
    Position = 0.3
    TriggerEventBufferSize = 10
    BarrierFunctionality = Off
  ProcessPoint[3]:
    Name = PP3
    SectorRef = SubSector1_3
    Position = 0.66
    TriggerEventBufferSize = 10
    BarrierFunctionality = Off
  ProcessPoint[4]:
    Name = PP4
    SectorRef = SubSector1_4
    Position = 0.4
    TriggerEventBufferSize = 10
    BarrierFunctionality = On
  ProcessPoint[5]:
    Name = PB2
    SectorRef = SubSector2_1
    PositionRelativeTo = FromEnd
    TriggerEventBufferSize = 10
    BarrierFunctionality = On
  ProcessPoint[6]:
    Name = PB3
    SectorRef = SubSector3_1
    PositionRelativeTo = FromEnd
    TriggerEventBufferSize = 10
    BarrierFunctionality = On
  ProcessPoint[7]:
    Name = PP5
    SectorRef = SubSector1_4
    Position = 0.34
    TriggerEventBufferSize = 10
    BarrierFunctionality = Off
  ProcessPoint[8]:
    Name = PP6
    SectorRef = SubSector1_2
    TriggerEventBufferSize = 10
    BarrierFunctionality = Off
```

### Config_5.assemblyfeature - 5PC900_TS17_00/mappMotion/Config_5.assemblyfeature
```
Element AssemblyFeature_1 (Type=assemblyfeature)
  Type = InitShuttleSim
    InitShuttleSim[1]:
      SectorRef = SectorTrack1
      Orientation = Positive
      ShuttleDefinition = ShuttleSetDefinition
        StartPosition = 2.0
        NumberOfShuttles = 15
        DistnaceBetweenShuttles = 0.15
    InitShuttleSim[2]:
      SectorRef = SectorTrack2
      Orientation = Negative
      ShuttleDefinition = ShuttleSetDefinition
        StartPosition = 0.1
        NumberOfShuttles = 5
        DistnaceBetweenShuttles = 0.15
    InitShuttleSim[3]:
      SectorRef = SectorTrack3
      Orientation = Negative
      ShuttleDefinition = ShuttleSetDefinition
        StartPosition = 0.1
        NumberOfShuttles = 5
        DistnaceBetweenShuttles = 0.15
    InitShuttleSim[4]:
      SectorRef = SectorTrack4
      Orientation = Negative
      ShuttleDefinition = ShuttleSetDefinition
        StartPosition = 0.1
        NumberOfShuttles = 5
        DistnaceBetweenShuttles = 0.15
    InitShuttleSim[5]:
      SectorRef = SectorTrack6
      Orientation = Positive
      ShuttleDefinition = ShuttleSetDefinition
        StartPosition = 0.1
        NumberOfShuttles = 3
        DistnaceBetweenShuttles = 0.15
Element AssemblyFeature_2 (Type=assemblyfeature)
  Type = ShtSectorAutoAttach
    Priority[1]:
      SectorRef = SectorTrack1
      Orientation = Positive
    Priority[2]:
      SectorRef = SectorTrack2
      Orientation = Negative
    Priority[3]:
      SectorRef = SectorTrack3
      Orientation = Negative
    Priority[4]:
      SectorRef = SectorTrack4
      Orientation = Negative
    Priority[5]:
      SectorRef = SectorTrack5
      Orientation = Negative
    Priority[6]:
      SectorRef = SectorTrack6
      Orientation = Positive
```

## Logical view

Binary libraries used (declarations not repeated): operator, runtime, astime, AsIecCon, AsZip, FileIO, brsystem, AsSem, sys_lib, AsBrStr, AsIODiag, DataObj, AsXml, standard, McBase 5.09.2, McAcpAx 5.11.3, McAcpTrak 5.11.3, McAxis 5.09.2, MpAxis 5.11.3, MpBase 5.09.0, MpAlarmX 5.09.1, CoTrace

### Global.typ - Global data types
```iecst
(*shuttle-UserData structure*)

TYPE
	ShuttleUserData_typ : 	STRUCT
		Task : ShuttleTask_enum;
		Partnumber : UDINT; (*example: product part number*)
		State : ShuttleState_enum;
	END_STRUCT;
	ShuttleTask_enum :
		(
		NoTask,
		PartsToCell1,
		PartsFromCell1,
		PartsToCell2,
		PartsFromCell2,
		MoveSubAssembly,
		MoveAssembly
		);
	ShuttleState_enum :
		(
		WaitingNewCommand,
		StartingProcess,
		InProcess,
		InPosition
		);
END_TYPE

(*Assembly Interface Type*)

TYPE
	TrakAsmCommand_type : 	STRUCT
		Power : BOOL;
		ShuttleStart : BOOL;
		ShuttleStop : {REDUND_UNREPLICABLE} BOOL;
	END_STRUCT;
	TrakAsmParameter_type : 	STRUCT
		Velocity : REAL;
		Acceleration : REAL;
		Deceleration : REAL;
	END_STRUCT;
	TrakAsmStatus_type : 	STRUCT
		Disabled : BOOL;
		Ready : BOOL;
		Homing : BOOL;
		Stopping : BOOL;
		ErrorStop : BOOL;
	END_STRUCT;
	TrakAsm_type : 	STRUCT
		Command : TrakAsmCommand_type;
		Parameter : TrakAsmParameter_type;
		Status : TrakAsmStatus_type;
	END_STRUCT;
END_TYPE
```

### Global.var - Global variables
```iecst
(*Assembly interface*)
VAR
	HMITaskCompleteCell2 : BOOL;
	HMITaskCompleteCell1 : BOOL;
	AddJob : BOOL;
	EmptyFixtureCell1 : INT;
	EmptyFixtureCell1Bool : BOOL;
	EmptyFixtureCell2 : INT;
	EmptyFixtureCell2Bool : BOOL;
END_VAR
(*shuttle monitor structure for Vis*)
VAR
	gShuttleMon : McAcpTrakAssemblyMonData;
END_VAR
(*shuttle-UserData structure*)
VAR
	gShuttleUserData : ShuttleUserData_typ;
	gTrakAsm : TrakAsm_type;
	HMILoadOffTrack : BOOL;
	LoadOffTrack : BOOL;
	HMILoadOnTrack : BOOL;
	LoadOnTrack : BOOL;
	Locked : BOOL;
	MoveAssemblyBool : BOOL;
	MoveAssemblyPart : INT;
	MoveSubAssemblyPartBool : BOOL;
	MoveSubAssemblyPart : INT;
	NeedPartCell1 : INT;
	NeedPartcell1Bool : BOOL;
	NeedPartCell2 : INT;
	NeedPartCell2Bool : BOOL;
	Ok : BOOL;
	OutletBarrierLocked : BOOL;
	Safety_Status : STRING[80];
	Status_hmi : STRING[80];
	TaskCompleteCell1 : BOOL;
	TaskCompleteCell2 : BOOL;
	Track5_Occupied : BOOL;
	Track6_Occupied : BOOL;
	TriggerCount : BOOL;
	WaitingBarrier : BOOL;
	WaitingLoadOff : BOOL;
	WaitingLoadOn : BOOL;
	Reset : BOOL;
	WaitingCell1 : BOOL;
	WaitingCell2 : BOOL;
END_VAR
```

- AS4_HW_8YF1I01.AB2B.00-1.exe (binary file, 157097 bytes)
### Program Logical/StartMovement (IEC)

#### Types.typ
```iecst
TYPE
	StepEnum :
		(
		POWER_OFF,
		POWER_ON,
		ADD_SHUTTLE,
		GET_SHUTTLE,
		READY,
		PROCESS,
		STOPPING,
		RESET
		);
	SubStepEnum :
		(
		GetShuttles,
		Userdata_Set,
		Userdata_Get,
		Reset_Process
		);
END_TYPE
```

#### Variables.var
```iecst
(*constants*)
VAR
	Status : STRING[80];
	PowerOffTrack2 : BOOL;
	MC_BR_SegPowerOff_AcpTrak_9 : MC_BR_SegPowerOff_AcpTrak;
	MC_BR_SegPowerOff_AcpTrak_8 : MC_BR_SegPowerOff_AcpTrak;
	MC_BR_SegPowerOff_AcpTrak_7 : MC_BR_SegPowerOff_AcpTrak;
	MC_BR_SegPowerOff_AcpTrak_6 : MC_BR_SegPowerOff_AcpTrak;
	MC_BR_SegPowerOff_AcpTrak_5 : MC_BR_SegPowerOff_AcpTrak;
	MC_BR_SegPowerOff_AcpTrak_4 : MC_BR_SegPowerOff_AcpTrak;
	MC_BR_SegPowerOff_AcpTrak_3 : MC_BR_SegPowerOff_AcpTrak;
	MC_BR_SegPowerOff_AcpTrak_2 : MC_BR_SegPowerOff_AcpTrak;
	MC_BR_SegPowerOff_AcpTrak_1 : MC_BR_SegPowerOff_AcpTrak;
	MC_BR_SegPowerOn_AcpTrak_9 : MC_BR_SegPowerOn_AcpTrak;
	MC_BR_SegPowerOn_AcpTrak_8 : MC_BR_SegPowerOn_AcpTrak;
	MC_BR_SegPowerOn_AcpTrak_7 : MC_BR_SegPowerOn_AcpTrak;
	MC_BR_SegPowerOn_AcpTrak_6 : MC_BR_SegPowerOn_AcpTrak;
	MC_BR_SegPowerOn_AcpTrak_5 : MC_BR_SegPowerOn_AcpTrak;
	MC_BR_SegPowerOn_AcpTrak_4 : MC_BR_SegPowerOn_AcpTrak;
	MC_BR_SegPowerOn_AcpTrak_3 : MC_BR_SegPowerOn_AcpTrak;
	MC_BR_SegPowerOn_AcpTrak_2 : MC_BR_SegPowerOn_AcpTrak;
	MC_BR_SegPowerOn_AcpTrak_1 : MC_BR_SegPowerOn_AcpTrak;
	MC_BR_SegPowerOn_AcpTrak_0 : MC_BR_SegPowerOn_AcpTrak;
	MC_BR_SegPowerOff_AcpTrak_0 : MC_BR_SegPowerOff_AcpTrak;
END_VAR
VAR CONSTANT
	NUM_SIM_SHUTTLES : USINT := 4; (*Maximum Shuttles Added in the Simulation*)
	MAX_NUM_SHUTTLES : USINT := 40; (*Maximum Shuttles Handled by the Trak*)
END_VAR
(*add shuttles for simulation*)
VAR
	SimShuttlePosition : ARRAY[1..MAX_NUM_SHUTTLES] OF LREAL;
END_VAR
(*sequence control*)
VAR
	Step : StepEnum;
	SubStep : SubStepEnum;
	CntShuttle : UINT;
	CntReset : UINT;
	ShuttleAxis : ARRAY[1..MAX_NUM_SHUTTLES] OF McAxisType;
	i : INT;
END_VAR
(*FUB*)
VAR
	MC_BR_AsmPowerOn_AcpTrak_0 : MC_BR_AsmPowerOn_AcpTrak;
	MC_BR_AsmPowerOff_AcpTrak_0 : MC_BR_AsmPowerOff_AcpTrak;
	ShuttleUserData : ShuttleUserData_typ;
	MC_BR_SecAddShuttle_AcpTrak_0 : MC_BR_SecAddShuttle_AcpTrak;
	MC_BR_AsmGetShuttle_AcpTrak_0 : MC_BR_AsmGetShuttle_AcpTrak;
	MC_BR_RoutedMoveVel_AcpTrak_0 : MC_BR_RoutedMoveVel_AcpTrak;
	MC_Stop_0 : MC_Stop;
	MC_BR_AsmReadStatus_AcpTrak_0 : MC_BR_AsmReadStatus_AcpTrak;
	SizeofUserdata : UDINT;
	MC_BR_AsmReset_AcpTrak_0 : MC_BR_AsmReset_AcpTrak;
	Shuttles_exist : BOOL;
	HMI_Start : BOOL;
	HMI_stop : BOOL;
	MC_BR_ShCopyUserData_AcpTrak_0 : MC_BR_ShCopyUserData_AcpTrak;
END_VAR
```

#### Main.st
```iecst
PROGRAM _INIT
    (* Set Shuttlepositions for Simulation (Starting at Position 0 on specified Sector) *)
	FOR i := 1 TO NUM_SIM_SHUTTLES DO
		SimShuttlePosition[i] := 0.15 * (i - 1);
	END_FOR

	(* Init Parameters for Shuttle movements *)
	gTrakAsm.Parameter.Velocity := 0.5;
	gTrakAsm.Parameter.Acceleration := 20;
	gTrakAsm.Parameter.Deceleration := 20;

	(* Write this value into the Size of Userdata in the Shuttle Stereotype configuration *)
	SizeofUserdata := SIZEOF(gShuttleUserData);

	(* Assembly reference for FUB's *)
	MC_BR_AsmPowerOn_AcpTrak_0.Assembly     := ADR(gAssembly_1);
	MC_BR_AsmGetShuttle_AcpTrak_0.Assembly  := ADR(gAssembly_1);
	MC_BR_AsmPowerOff_AcpTrak_0.Assembly    := ADR(gAssembly_1);
	MC_BR_AsmReadStatus_AcpTrak_0.Assembly  := ADR(gAssembly_1);
	MC_BR_AsmReset_AcpTrak_0.Assembly       := ADR(gAssembly_1);

	(* Enable reading of current status of the assembly *)
	MC_BR_AsmReadStatus_AcpTrak_0.Enable := TRUE;
    CntReset := 1;
END_PROGRAM

PROGRAM _CYCLIC

	IF HMI_Start THEN
		gTrakAsm.Command.Power := TRUE;
	END_IF

	IF HMI_stop THEN
		gTrakAsm.Command.Power := FALSE;
	END_IF

	CASE Step OF

			(*        Assemply power off and waiting for power on command        *)
		POWER_OFF:
			Status := 'Power Off';
			IF EDGEPOS(MC_BR_AsmPowerOff_AcpTrak_0.Done) THEN    (* When power off is done, delete the shuttle reference *)
				MC_BR_AsmPowerOff_AcpTrak_0.Execute := FALSE;
				brsmemset(ADR(ShuttleAxis), 0, SIZEOF(ShuttleAxis));
			ELSIF NOT(gTrakAsm.Status.Disabled) THEN             (* Assembly is not powered off yet *)
				MC_BR_AsmPowerOff_AcpTrak_0.Execute := TRUE;
			ELSIF (gTrakAsm.Command.Power) THEN
				Step := POWER_ON;
			END_IF

			(*        Assembly power ON        *)
		POWER_ON:
			Status := 'Power On';
			MC_BR_AsmPowerOn_AcpTrak_0.Execute := TRUE;

			IF EDGEPOS(MC_BR_AsmPowerOn_AcpTrak_0.Done)THEN
				CntShuttle := 1;
				IF NOT DiagCpuIsARsim() THEN
					Step := GET_SHUTTLE;
				ELSIF NOT(Shuttles_exist) THEN
					Step := ADD_SHUTTLE;
				ELSE
					Step := READY;
				END_IF
			END_IF
			(*        Adding Shuttles for simulation (These steps are not needed on real Hardware)        *)
		ADD_SHUTTLE:
			Status := 'Add_Shuttle';
			IF (MC_BR_SecAddShuttle_AcpTrak_0.Done) THEN
				CntShuttle := CntShuttle + 1;
			ELSIF (CntShuttle <= NUM_SIM_SHUTTLES) THEN
				MC_BR_SecAddShuttle_AcpTrak_0.Sector   := ADR(SectorTrack1);
				MC_BR_SecAddShuttle_AcpTrak_0.Execute  := TRUE;
				MC_BR_SecAddShuttle_AcpTrak_0.Position := SimShuttlePosition[CntShuttle];
				MC_BR_SecAddShuttle_AcpTrak_0.AdvancedParameters.Velocity := 0.0;
			ELSE
				CntShuttle := 1;
				Step := GET_SHUTTLE;
			END_IF

			(*        Get all available on the assembly (physically available on the real hardware or the added ones in the simulation)        *)
		GET_SHUTTLE:
			Status := 'Get_Shuttle';
			MC_BR_AsmGetShuttle_AcpTrak_0.Enable := TRUE;

			IF (MC_BR_AsmGetShuttle_AcpTrak_0.Valid) THEN
				IF (MC_BR_AsmGetShuttle_AcpTrak_0.RemainingCount <> (MC_BR_AsmGetShuttle_AcpTrak_0.TotalCount - CntShuttle)) THEN
					CntShuttle := CntShuttle + 1;
					MC_BR_AsmGetShuttle_AcpTrak_0.Next := FALSE;
				ELSE
					ShuttleAxis[CntShuttle] := MC_BR_AsmGetShuttle_AcpTrak_0.Axis;    (*Save all Axis References to an array for global movement commands*)
					MC_BR_AsmGetShuttle_AcpTrak_0.Next := TRUE;   (*Get next Shuttle reference with positive Edge on .next*)

					IF (MC_BR_AsmGetShuttle_AcpTrak_0.RemainingCount = 0) THEN
						MC_BR_AsmGetShuttle_AcpTrak_0.Enable := FALSE;
						MC_BR_AsmGetShuttle_AcpTrak_0.Next := FALSE;
						Shuttles_exist := TRUE;
						Step := READY;
					END_IF
				END_IF
			END_IF

			(*        Assembly Active and ready for movement        *)
		READY:
			Status := 'Ready';
			IF (gTrakAsm.Command.Power = FALSE) THEN     (*Power Off Command*)
				Step := POWER_OFF;
			ELSIF (gTrakAsm.Command.ShuttleStart) THEN   (*Waiting for Movement command*)
				gTrakAsm.Command.ShuttleStart := FALSE;
				CntShuttle := 1;
				CntReset := 1;
				Step := PROCESS;
			END_IF

			(*             Accelerate all shuttles in assembly via the same target position to the same velocity            *)
			(* Used for startup, to accelerate all shuttles to an initial velocity in order to pass the first process-point *)
		PROCESS:
			Status := 'Process';
			IF EDGEPOS(MC_BR_RoutedMoveVel_AcpTrak_0.Active) THEN
				CntShuttle := CntShuttle + 1;
				MC_BR_RoutedMoveVel_AcpTrak_0.Execute := FALSE;
			ELSIF (CntShuttle > 0) THEN
				IF (ShuttleAxis[CntShuttle].controlif <> 0) THEN
					MC_BR_RoutedMoveVel_AcpTrak_0.Axis          := ADR(ShuttleAxis[CntShuttle]);
					MC_BR_RoutedMoveVel_AcpTrak_0.Execute       := TRUE;

					MC_BR_RoutedMoveVel_AcpTrak_0.Sector        := ADR(SectorTrack1);
					MC_BR_RoutedMoveVel_AcpTrak_0.Position      := SimShuttlePosition[NUM_SIM_SHUTTLES] + 0.15;
					MC_BR_RoutedMoveVel_AcpTrak_0.Velocity      := gTrakAsm.Parameter.Velocity;
					MC_BR_RoutedMoveVel_AcpTrak_0.RouteVelocity := gTrakAsm.Parameter.Velocity;
					MC_BR_RoutedMoveVel_AcpTrak_0.Acceleration  := gTrakAsm.Parameter.Acceleration;
					MC_BR_RoutedMoveVel_AcpTrak_0.Deceleration  := gTrakAsm.Parameter.Deceleration;
					MC_BR_RoutedMoveVel_AcpTrak_0.Jerk          := 0.0;
					MC_BR_RoutedMoveVel_AcpTrak_0.BufferMode    := mcABORTING;
					MC_BR_RoutedMoveVel_AcpTrak_0.AdvancedParameters.StartDirection     := mcDIR_UNDEFINED;
					MC_BR_RoutedMoveVel_AcpTrak_0.AdvancedParameters.EndDirection       := mcDIR_POSITIVE;
					MC_BR_RoutedMoveVel_AcpTrak_0.AdvancedParameters.ShuttleOrientation := mcDIR_UNDEFINED;
				END_IF
			 END_IF

			CASE SubStep OF
				GetShuttles:
					IF EDGEPOS (Reset) THEN

						IF WaitingCell1 THEN
							TaskCompleteCell1 := TRUE;
						END_IF
						IF WaitingCell2 THEN
							TaskCompleteCell2 := TRUE;
						END_IF
						IF WaitingLoadOn THEN
							LoadOnTrack := TRUE;
						END_IF
						IF WaitingLoadOff THEN
							LoadOffTrack := TRUE;
						END_IF
						MC_BR_AsmGetShuttle_AcpTrak_0.Enable := TRUE;
					END_IF

					IF (MC_BR_AsmGetShuttle_AcpTrak_0.Valid) THEN
						IF (MC_BR_AsmGetShuttle_AcpTrak_0.RemainingCount <> 0) AND MC_BR_AsmGetShuttle_AcpTrak_0.Next THEN
								MC_BR_AsmGetShuttle_AcpTrak_0.Next := FALSE;
							ELSE
								ShuttleAxis[CntReset] := MC_BR_AsmGetShuttle_AcpTrak_0.Axis;    (*Save all Axis References to an array for global movement commands*)
								MC_BR_AsmGetShuttle_AcpTrak_0.Next := TRUE;   (*Get next Shuttle reference with positive Edge on .next*)
								CntReset := CntReset+1;
								SubStep := Userdata_Get;
								IF (MC_BR_AsmGetShuttle_AcpTrak_0.RemainingCount = 0) THEN
									MC_BR_AsmGetShuttle_AcpTrak_0.Enable := FALSE;
									MC_BR_AsmGetShuttle_AcpTrak_0.Next := FALSE;
									CntReset := 1;
									Reset := FALSE;
								END_IF
							END_IF
					END_IF

					Userdata_Get:
						(* The userdata is copied on a local variable *)
						MC_BR_ShCopyUserData_AcpTrak_0.Axis := ADR(ShuttleAxis[CntReset]);
						MC_BR_ShCopyUserData_AcpTrak_0.Execute := TRUE;
						MC_BR_ShCopyUserData_AcpTrak_0.DataAddress := ADR(ShuttleUserData);
						MC_BR_ShCopyUserData_AcpTrak_0.DataSize := SIZEOF(ShuttleUserData);
						MC_BR_ShCopyUserData_AcpTrak_0.Mode := mcACPTRAK_USERDATA_GET;
						(* After copying go to the next step *)

						IF EDGEPOS(MC_BR_ShCopyUserData_AcpTrak_0.Done) THEN
							MC_BR_ShCopyUserData_AcpTrak_0.Execute := FALSE;
							SubStep := Reset_Process;
						END_IF

					Reset_Process:

					ShuttleUserData.Task := NoTask;
						SubStep := Userdata_Set;

						Userdata_Set:
							(* The modified userdata will be copied back on the shuttle *)
							MC_BR_ShCopyUserData_AcpTrak_0.Axis := ADR(ShuttleAxis[CntReset]);
							MC_BR_ShCopyUserData_AcpTrak_0.Execute := TRUE;
							MC_BR_ShCopyUserData_AcpTrak_0.DataAddress := ADR(ShuttleUserData);
							MC_BR_ShCopyUserData_AcpTrak_0.DataSize := SIZEOF(ShuttleUserData);
							MC_BR_ShCopyUserData_AcpTrak_0.Mode := mcACPTRAK_USERDATA_SET;

							(* After copying go to the first step and wait for new event *)
							IF EDGEPOS(MC_BR_ShCopyUserData_AcpTrak_0.Done) THEN
								MC_BR_ShCopyUserData_AcpTrak_0.Execute := FALSE;
								SubStep := GetShuttles;

							END_IF
					END_CASE

			IF PowerOffTrack2 THEN

				MC_BR_SegPowerOff_AcpTrak_0.Execute := TRUE;
				MC_BR_SegPowerOff_AcpTrak_1.Execute := TRUE;
				MC_BR_SegPowerOff_AcpTrak_2.Execute := TRUE;
//				MC_BR_SegPowerOff_AcpTrak_3.Execute := TRUE;
				MC_BR_SegPowerOff_AcpTrak_4.Execute := TRUE;
				MC_BR_SegPowerOff_AcpTrak_5.Execute := TRUE;
				MC_BR_SegPowerOff_AcpTrak_6.Execute := TRUE;
				MC_BR_SegPowerOff_AcpTrak_7.Execute := TRUE;
				MC_BR_SegPowerOff_AcpTrak_8.Execute := TRUE;
				MC_BR_SegPowerOff_AcpTrak_9.Execute := TRUE;
				MC_BR_SegPowerOn_AcpTrak_0.Execute := FALSE;
				MC_BR_SegPowerOn_AcpTrak_1.Execute := FALSE;
				MC_BR_SegPowerOn_AcpTrak_2.Execute := FALSE;
				MC_BR_SegPowerOn_AcpTrak_3.Execute := FALSE;
				MC_BR_SegPowerOn_AcpTrak_4.Execute := FALSE;
				MC_BR_SegPowerOn_AcpTrak_5.Execute := FALSE;
				MC_BR_SegPowerOn_AcpTrak_6.Execute := FALSE;
				MC_BR_SegPowerOn_AcpTrak_7.Execute := FALSE;
				MC_BR_SegPowerOn_AcpTrak_8.Execute := FALSE;
				MC_BR_SegPowerOn_AcpTrak_9.Execute := FALSE;
				MC_BR_SegPowerOff_AcpTrak_0.Segment := ADR(SEG_2_74);
				MC_BR_SegPowerOff_AcpTrak_1.Segment := ADR(SEG_2_75);
				MC_BR_SegPowerOff_AcpTrak_2.Segment := ADR(SEG_2_76);
//				MC_BR_SegPowerOff_AcpTrak_3.Segment := ADR(SEG_2_77);
				MC_BR_SegPowerOff_AcpTrak_4.Segment := ADR(SEG_2_78);
				MC_BR_SegPowerOff_AcpTrak_5.Segment := ADR(SEG_2_79);
				MC_BR_SegPowerOff_AcpTrak_6.Segment := ADR(SEG_2_80);
				MC_BR_SegPowerOff_AcpTrak_7.Segment := ADR(SEG_2_81);
				MC_BR_SegPowerOff_AcpTrak_8.Segment := ADR(SEG_2_82);
				MC_BR_SegPowerOff_AcpTrak_9.Segment := ADR(SEG_2_83);

			ELSIF MC_BR_SegPowerOff_AcpTrak_0.Execute AND NOT PowerOffTrack2 THEN

				MC_BR_SegPowerOn_AcpTrak_0.Execute := TRUE;
				MC_BR_SegPowerOn_AcpTrak_1.Execute := TRUE;
				MC_BR_SegPowerOn_AcpTrak_2.Execute := TRUE;
//				MC_BR_SegPowerOn_AcpTrak_3.Execute := TRUE;
				MC_BR_SegPowerOn_AcpTrak_4.Execute := TRUE;
				MC_BR_SegPowerOn_AcpTrak_5.Execute := TRUE;
				MC_BR_SegPowerOn_AcpTrak_6.Execute := TRUE;
				MC_BR_SegPowerOn_AcpTrak_7.Execute := TRUE;
				MC_BR_SegPowerOn_AcpTrak_8.Execute := TRUE;
				MC_BR_SegPowerOn_AcpTrak_9.Execute := TRUE;
				MC_BR_SegPowerOff_AcpTrak_0.Execute := FALSE;
				MC_BR_SegPowerOff_AcpTrak_1.Execute := FALSE;
				MC_BR_SegPowerOff_AcpTrak_2.Execute := FALSE;
				MC_BR_SegPowerOff_AcpTrak_3.Execute := FALSE;
				MC_BR_SegPowerOff_AcpTrak_4.Execute := FALSE;
				MC_BR_SegPowerOff_AcpTrak_5.Execute := FALSE;
				MC_BR_SegPowerOff_AcpTrak_6.Execute := FALSE;
				MC_BR_SegPowerOff_AcpTrak_7.Execute := FALSE;
				MC_BR_SegPowerOff_AcpTrak_8.Execute := FALSE;
				MC_BR_SegPowerOff_AcpTrak_9.Execute := FALSE;
				MC_BR_SegPowerOn_AcpTrak_0.Segment := ADR(SEG_2_74);
				MC_BR_SegPowerOn_AcpTrak_1.Segment := ADR(SEG_2_75);
				MC_BR_SegPowerOn_AcpTrak_2.Segment := ADR(SEG_2_76);
//				MC_BR_SegPowerOn_AcpTrak_3.Segment := ADR(SEG_2_77);
				MC_BR_SegPowerOn_AcpTrak_4.Segment := ADR(SEG_2_78);
				MC_BR_SegPowerOn_AcpTrak_5.Segment := ADR(SEG_2_79);
				MC_BR_SegPowerOn_AcpTrak_6.Segment := ADR(SEG_2_80);
				MC_BR_SegPowerOn_AcpTrak_7.Segment := ADR(SEG_2_81);
				MC_BR_SegPowerOn_AcpTrak_7.Segment := ADR(SEG_2_82);
				MC_BR_SegPowerOn_AcpTrak_9.Segment := ADR(SEG_2_83);

			END_IF

			IF(gTrakAsm.Command.ShuttleStop) AND (CntShuttle > NUM_SIM_SHUTTLES) THEN   (*Waiting for Stop command*)
				CntShuttle := 1;
				Step := STOPPING;
			END_IF

			(* When there is invalid speed or acceleration setting, or shuttle caused ErrorStop *)
			IF (MC_BR_RoutedMoveVel_AcpTrak_0.Error) THEN
				MC_BR_AsmReset_AcpTrak_0.Execute := TRUE;
				Step := RESET;
			END_IF

			(*        Stop all Shuttles with specified Deceleration at their current location        *)
		STOPPING:
			Status := 'Stopping';
			IF EDGEPOS(MC_Stop_0.Done) THEN
				CntShuttle := CntShuttle + 1;
				MC_Stop_0.Execute := FALSE;
			ELSIF (ShuttleAxis[CntShuttle].controlif <> 0) AND NOT(MC_Stop_0.Busy) THEN
				MC_Stop_0.Axis         := ADR(ShuttleAxis[CntShuttle]);
				MC_Stop_0.Execute      := TRUE;
				MC_Stop_0.Deceleration := 20;
				MC_Stop_0.Jerk         := 0.0;
				MC_BR_RoutedMoveVel_AcpTrak_0.Execute := FALSE;
			END_IF

			IF EDGEPOS(MC_Stop_0.Done) AND (CntShuttle > NUM_SIM_SHUTTLES) THEN (* Back to ready, after every shuttle on the trak has stopped *)
				gTrakAsm.Command.ShuttleStop := FALSE;
				Step := READY;
			END_IF

			(*        Reset Assembly due to an error        *)
		RESET:
			Status := 'Reset';
			IF EDGEPOS(MC_BR_AsmReset_AcpTrak_0.Done) THEN
				gTrakAsm.Command.ShuttleStart    := FALSE;
				gTrakAsm.Command.ShuttleStop     := FALSE;
				MC_BR_AsmReset_AcpTrak_0.Execute := FALSE;
				MC_BR_RoutedMoveVel_AcpTrak_0.Execute := FALSE;

				Step := READY;
			END_IF

	END_CASE

	(* Read Assembly status cyclic to Assembly interface *)
	gTrakAsm.Status.Disabled  := MC_BR_AsmReadStatus_AcpTrak_0.AssemblyDisabled;
	gTrakAsm.Status.Ready     := MC_BR_AsmReadStatus_AcpTrak_0.AssemblyReady;
	gTrakAsm.Status.Homing    := MC_BR_AsmReadStatus_AcpTrak_0.AssemblyHoming;
	gTrakAsm.Status.Stopping  := MC_BR_AsmReadStatus_AcpTrak_0.AssemblyStopping;
	gTrakAsm.Status.ErrorStop := MC_BR_AsmReadStatus_AcpTrak_0.AssemblyErrorStop;

	(*        Cyclic FUB call        *)
	MC_BR_AsmPowerOn_AcpTrak_0();
	MC_BR_AsmPowerOn_AcpTrak_0.Execute := FALSE;
	MC_BR_SecAddShuttle_AcpTrak_0();
	MC_BR_SecAddShuttle_AcpTrak_0.Execute := FALSE;
	MC_BR_AsmGetShuttle_AcpTrak_0();
	MC_BR_AsmPowerOff_AcpTrak_0();
	MC_BR_RoutedMoveVel_AcpTrak_0();
	MC_Stop_0();
	MC_BR_AsmReadStatus_AcpTrak_0();
	MC_BR_AsmReset_AcpTrak_0();
	MC_BR_SegPowerOff_AcpTrak_0();
	MC_BR_SegPowerOff_AcpTrak_1();
	MC_BR_SegPowerOff_AcpTrak_2();
	MC_BR_SegPowerOff_AcpTrak_3();
	MC_BR_SegPowerOff_AcpTrak_4();
	MC_BR_SegPowerOff_AcpTrak_5();
	MC_BR_SegPowerOff_AcpTrak_6();
	MC_BR_SegPowerOff_AcpTrak_7();
	MC_BR_SegPowerOff_AcpTrak_8();
	MC_BR_SegPowerOff_AcpTrak_9();
	MC_BR_SegPowerOn_AcpTrak_0();
	MC_BR_SegPowerOn_AcpTrak_1();
	MC_BR_SegPowerOn_AcpTrak_2();
	MC_BR_SegPowerOn_AcpTrak_3();
	MC_BR_SegPowerOn_AcpTrak_4();
	MC_BR_SegPowerOn_AcpTrak_5();
	MC_BR_SegPowerOn_AcpTrak_6();
	MC_BR_SegPowerOn_AcpTrak_7();
	MC_BR_SegPowerOn_AcpTrak_8();
	MC_BR_SegPowerOn_AcpTrak_9();
	MC_BR_ShCopyUserData_AcpTrak_0();

	IF EmptyFixtureCell1 = 1 AND EmptyFixtureCell2 = 1 AND NeedPartCell1 = 1 AND NeedPartCell2 = 1 AND MoveAssemblyPart = 1 AND TaskCompleteCell1 AND TaskCompleteCell2 AND LoadOnTrack AND LoadOffTrack THEN
		Ok := TRUE;
	END_IF

END_PROGRAM
```

### Program Logical/Vis (IEC)

#### Variables.var
```iecst
VAR
	i : USINT := 0;
	NumVisShuttle : USINT := 0;
	pUserData : REFERENCE TO ShuttleUserData_typ;
	Shuttle0_Angel : REAL;
	Shuttle0_X : REAL;
	Shuttle0_Y : REAL;
	Shuttle1_Angel : REAL;
	Shuttle1_X : REAL;
	Shuttle1_Y : REAL;
	Shuttle2_Angel : REAL;
	Shuttle2_X : REAL;
	Shuttle2_Y : REAL;
	Shuttle3_Angel : REAL;
	Shuttle3_X : REAL;
	Shuttle3_Y : REAL;
	Shuttle4_Angel : REAL;
	Shuttle4_X : REAL;
	Shuttle4_Y : REAL;
	Shuttle5_Angel : REAL;
	Shuttle5_X : REAL;
	Shuttle5_Y : REAL;
	Shuttle6_Angel : REAL;
	Shuttle6_X : REAL;
	Shuttle6_Y : REAL;
	Shuttle7_Angel : REAL;
	Shuttle7_X : REAL;
	Shuttle7_Y : REAL;
	Shuttle8_Angel : REAL;
	Shuttle8_X : REAL;
	Shuttle8_Y : REAL;
	Shuttle9_Angel : REAL;
	Shuttle9_X : REAL;
	Shuttle9_Y : REAL;
	Shuttle10_Angel : REAL;
	Shuttle10_X : REAL;
	Shuttle10_Y : REAL;
	Shuttle11_Angel : REAL;
	Shuttle11_X : REAL;
	Shuttle11_Y : REAL;
	Shuttle12_Angel : REAL;
	Shuttle12_X : REAL;
	Shuttle12_Y : REAL;
	Shuttle13_Angel : REAL;
	Shuttle13_X : REAL;
	Shuttle13_Y : REAL;
	Shuttle14_Angel : REAL;
	Shuttle44_Angel : REAL;
	Shuttle14_X : REAL;
	Shuttle14_Y : REAL;
	Shuttle15_Angel : REAL;
	Shuttle15_X : REAL;
	Shuttle15_Y : REAL;
	Shuttle16_Angel : REAL;
	Shuttle16_X : REAL;
	Shuttle16_Y : REAL;
	Shuttle17_Angel : REAL;
	Shuttle17_X : REAL;
	Shuttle17_Y : REAL;
	Shuttle18_Angel : REAL;
	Shuttle18_X : REAL;
	Shuttle18_Y : REAL;
	Shuttle19_Angel : REAL;
	Shuttle19_X : REAL;
	Shuttle19_Y : REAL;
	Shuttle20_Angel : REAL;
	Shuttle20_X : REAL;
	Shuttle20_Y : REAL;
	Shuttle21_Angel : REAL;
	Shuttle21_X : REAL;
	Shuttle21_Y : REAL;
	Shuttle22_Angel : REAL;
	Shuttle22_X : REAL;
	Shuttle22_Y : REAL;
	Shuttle23_Angel : REAL;
	Shuttle23_X : REAL;
	Shuttle23_Y : REAL;
	Shuttle24_Angel : REAL;
	Shuttle24_X : REAL;
	Shuttle24_Y : REAL;
	Shuttle25_Angel : REAL;
	Shuttle25_X : REAL;
	Shuttle25_Y : REAL;
	Shuttle26_Angel : REAL;
	Shuttle26_X : REAL;
	Shuttle26_Y : REAL;
	Shuttle27_Angel : REAL;
	Shuttle27_X : REAL;
	Shuttle27_Y : REAL;
	Shuttle28_Angel : REAL;
	Shuttle28_X : REAL;
	Shuttle28_Y : REAL;
	Shuttle29_Angel : REAL;
	Shuttle29_X : REAL;
	Shuttle29_Y : REAL;
	Shuttle30_Angel : REAL;
	Shuttle30_X : REAL;
	Shuttle30_Y : REAL;
	Shuttle31_Angel : REAL;
	Shuttle31_X : REAL;
	Shuttle31_Y : REAL;
	Shuttle32_Angel : REAL;
	Shuttle32_X : REAL;
	Shuttle32_Y : REAL;
	Shuttle33_Angel : REAL;
	Shuttle33_X : REAL;
	Shuttle33_Y : REAL;
	Shuttle34_Angel : REAL;
	Shuttle34_X : REAL;
	Shuttle34_Y : REAL;
	Shuttle35_Angel : REAL;
	Shuttle35_X : REAL;
	Shuttle35_Y : REAL;
	Shuttle36_Angel : REAL;
	Shuttle36_X : REAL;
	Shuttle36_Y : REAL;
	Shuttle37_Angel : REAL;
	Shuttle37_X : REAL;
	Shuttle37_Y : REAL;
	Shuttle38_Angel : REAL;
	Shuttle38_X : REAL;
	Shuttle38_Y : REAL;
	Shuttle39_Angel : REAL;
	Shuttle39_X : REAL;
	Shuttle39_Y : REAL;
	Shuttle40_Angel : REAL;
	Shuttle40_X : REAL;
	Shuttle40_Y : REAL;
	Shuttle41_Angel : REAL;
	Shuttle41_X : REAL;
	Shuttle41_Y : REAL;
	Shuttle42_Angel : REAL;
	Shuttle42_X : REAL;
	Shuttle42_Y : REAL;
	Shuttle43_Angel : REAL;
	Shuttle43_X : REAL;
	Shuttle43_Y : REAL;
	Shuttle44_X : REAL;
	Shuttle44_Y : REAL;
	SizeofVis : UDINT := 0;
	Vis : McAcpTrakAssemblyVisData;
END_VAR
```

#### Main.st
```iecst
PROGRAM _INIT

    // size of Vis structure - this value has to be entered in B&R scene viewer (PVI -> Options -> Size)
	SizeofVis := SIZEOF(Vis);
	// max number of displayed shuttles
	NumVisShuttle := SIZEOF(Vis.Shuttle) / SIZEOF(Vis.Shuttle[0]);
	//dummy call
	gShuttleMon;

END_PROGRAM

PROGRAM _CYCLIC

	FOR i:=0 TO (NumVisShuttle-1) DO
		IF gShuttleMon.Shuttle[i].Available THEN
			// format selected monitor data to fit B&R scene viewer
			Vis.Shuttle[i].Available     := 1;
			Vis.Shuttle[i].PositionX     := LREAL_TO_REAL(gShuttleMon.Shuttle[i].Position.X);
			Vis.Shuttle[i].PositionY     := LREAL_TO_REAL(gShuttleMon.Shuttle[i].Position.Y);
			Vis.Shuttle[i].RotationZ     := LREAL_TO_REAL(gShuttleMon.Shuttle[i].Orientation.Angle1);
			Vis.Shuttle[i].ExtentToFront := LREAL_TO_REAL(gShuttleMon.Shuttle[i].ExtentToFront);
			Vis.Shuttle[i].ExtentToBack  := LREAL_TO_REAL(gShuttleMon.Shuttle[i].ExtentToBack);
			Vis.Shuttle[i].Width         := LREAL_TO_REAL(gShuttleMon.Shuttle[i].Width);
			brsitoa(gShuttleMon.Shuttle[i].Index, ADR(Vis.Shuttle[i].Text));

			Shuttle0_X := LREAL_TO_REAL(gShuttleMon.Shuttle[0].Position.X);
			Shuttle0_Y := LREAL_TO_REAL(gShuttleMon.Shuttle[0].Position.Y);
			Shuttle0_Angel := LREAL_TO_REAL(gShuttleMon.Shuttle[0].Orientation.Angle1);
			Shuttle1_X := LREAL_TO_REAL(gShuttleMon.Shuttle[1].Position.X);
			Shuttle1_Y := LREAL_TO_REAL(gShuttleMon.Shuttle[1].Position.Y);
			Shuttle1_Angel := LREAL_TO_REAL(gShuttleMon.Shuttle[1].Orientation.Angle1);
			Shuttle2_X := LREAL_TO_REAL(gShuttleMon.Shuttle[2].Position.X);
			Shuttle2_Y := LREAL_TO_REAL(gShuttleMon.Shuttle[2].Position.Y);
			Shuttle2_Angel := LREAL_TO_REAL(gShuttleMon.Shuttle[2].Orientation.Angle1);
			Shuttle3_X := LREAL_TO_REAL(gShuttleMon.Shuttle[3].Position.X);
			Shuttle3_Y := LREAL_TO_REAL(gShuttleMon.Shuttle[3].Position.Y);
			Shuttle3_Angel := LREAL_TO_REAL(gShuttleMon.Shuttle[3].Orientation.Angle1);
			Shuttle4_X := LREAL_TO_REAL(gShuttleMon.Shuttle[4].Position.X);
			Shuttle4_Y := LREAL_TO_REAL(gShuttleMon.Shuttle[4].Position.Y);
			Shuttle4_Angel := LREAL_TO_REAL(gShuttleMon.Shuttle[4].Orientation.Angle1);
			Shuttle5_Angel := LREAL_TO_REAL(gShuttleMon.Shuttle[5].Orientation.Angle1);
			Shuttle5_X := LREAL_TO_REAL(gShuttleMon.Shuttle[5].Position.X);
			Shuttle5_Y := LREAL_TO_REAL(gShuttleMon.Shuttle[5].Position.Y);
			Shuttle6_Angel := LREAL_TO_REAL(gShuttleMon.Shuttle[6].Orientation.Angle1);
			Shuttle6_X := LREAL_TO_REAL(gShuttleMon.Shuttle[6].Position.X);
			Shuttle6_Y := LREAL_TO_REAL(gShuttleMon.Shuttle[6].Position.Y);
			Shuttle7_Angel := LREAL_TO_REAL(gShuttleMon.Shuttle[7].Orientation.Angle1);
			Shuttle7_X := LREAL_TO_REAL(gShuttleMon.Shuttle[7].Position.X);
			Shuttle7_Y := LREAL_TO_REAL(gShuttleMon.Shuttle[7].Position.Y);
			Shuttle8_Angel := LREAL_TO_REAL(gShuttleMon.Shuttle[8].Orientation.Angle1);
			Shuttle8_X := LREAL_TO_REAL(gShuttleMon.Shuttle[8].Position.X);
			Shuttle8_Y := LREAL_TO_REAL(gShuttleMon.Shuttle[8].Position.Y);
			Shuttle9_Angel := LREAL_TO_REAL(gShuttleMon.Shuttle[9].Orientation.Angle1);
			Shuttle9_X := LREAL_TO_REAL(gShuttleMon.Shuttle[9].Position.X);
			Shuttle9_Y := LREAL_TO_REAL(gShuttleMon.Shuttle[9].Position.Y);
			Shuttle10_Angel := LREAL_TO_REAL(gShuttleMon.Shuttle[10].Orientation.Angle1);
			Shuttle10_X := LREAL_TO_REAL(gShuttleMon.Shuttle[10].Position.X);
			Shuttle10_Y := LREAL_TO_REAL(gShuttleMon.Shuttle[10].Position.Y);
			Shuttle11_Angel := LREAL_TO_REAL(gShuttleMon.Shuttle[11].Orientation.Angle1);
			Shuttle11_X := LREAL_TO_REAL(gShuttleMon.Shuttle[11].Position.X);
			Shuttle11_Y := LREAL_TO_REAL(gShuttleMon.Shuttle[11].Position.Y);
			Shuttle12_Angel := LREAL_TO_REAL(gShuttleMon.Shuttle[12].Orientation.Angle1);
			Shuttle12_X := LREAL_TO_REAL(gShuttleMon.Shuttle[12].Position.X);
			Shuttle12_Y := LREAL_TO_REAL(gShuttleMon.Shuttle[12].Position.Y);
			Shuttle13_Angel := LREAL_TO_REAL(gShuttleMon.Shuttle[13].Orientation.Angle1);
			Shuttle13_X := LREAL_TO_REAL(gShuttleMon.Shuttle[13].Position.X);
			Shuttle13_Y := LREAL_TO_REAL(gShuttleMon.Shuttle[13].Position.Y);
			Shuttle14_Angel := LREAL_TO_REAL(gShuttleMon.Shuttle[14].Orientation.Angle1);
			Shuttle14_X := LREAL_TO_REAL(gShuttleMon.Shuttle[14].Position.X);
			Shuttle14_Y := LREAL_TO_REAL(gShuttleMon.Shuttle[14].Position.Y);
			Shuttle15_Angel := LREAL_TO_REAL(gShuttleMon.Shuttle[15].Orientation.Angle1);
			Shuttle15_X := LREAL_TO_REAL(gShuttleMon.Shuttle[15].Position.X);
			Shuttle15_Y := LREAL_TO_REAL(gShuttleMon.Shuttle[15].Position.Y);
			Shuttle16_Angel := LREAL_TO_REAL(gShuttleMon.Shuttle[16].Orientation.Angle1);
			Shuttle16_X := LREAL_TO_REAL(gShuttleMon.Shuttle[16].Position.X);
			Shuttle16_Y := LREAL_TO_REAL(gShuttleMon.Shuttle[16].Position.Y);
			Shuttle17_Angel := LREAL_TO_REAL(gShuttleMon.Shuttle[17].Orientation.Angle1);
			Shuttle17_X := LREAL_TO_REAL(gShuttleMon.Shuttle[17].Position.X);
			Shuttle17_Y := LREAL_TO_REAL(gShuttleMon.Shuttle[17].Position.Y);
			Shuttle18_Angel := LREAL_TO_REAL(gShuttleMon.Shuttle[18].Orientation.Angle1);
			Shuttle18_X := LREAL_TO_REAL(gShuttleMon.Shuttle[18].Position.X);
			Shuttle18_Y := LREAL_TO_REAL(gShuttleMon.Shuttle[18].Position.Y);
			Shuttle19_Angel := LREAL_TO_REAL(gShuttleMon.Shuttle[19].Orientation.Angle1);
			Shuttle19_X := LREAL_TO_REAL(gShuttleMon.Shuttle[19].Position.X);
			Shuttle19_Y := LREAL_TO_REAL(gShuttleMon.Shuttle[19].Position.Y);
			Shuttle20_Angel := LREAL_TO_REAL(gShuttleMon.Shuttle[20].Orientation.Angle1);
			Shuttle20_X := LREAL_TO_REAL(gShuttleMon.Shuttle[20].Position.X);
			Shuttle20_Y := LREAL_TO_REAL(gShuttleMon.Shuttle[20].Position.Y);
			Shuttle21_Angel := LREAL_TO_REAL(gShuttleMon.Shuttle[21].Orientation.Angle1);
			Shuttle21_X := LREAL_TO_REAL(gShuttleMon.Shuttle[21].Position.X);
			Shuttle21_Y := LREAL_TO_REAL(gShuttleMon.Shuttle[21].Position.Y);
			Shuttle22_Angel := LREAL_TO_REAL(gShuttleMon.Shuttle[22].Orientation.Angle1);
			Shuttle22_X := LREAL_TO_REAL(gShuttleMon.Shuttle[22].Position.X);
			Shuttle22_Y := LREAL_TO_REAL(gShuttleMon.Shuttle[22].Position.Y);
			Shuttle23_Angel := LREAL_TO_REAL(gShuttleMon.Shuttle[23].Orientation.Angle1);
			Shuttle23_X := LREAL_TO_REAL(gShuttleMon.Shuttle[23].Position.X);
			Shuttle23_Y := LREAL_TO_REAL(gShuttleMon.Shuttle[23].Position.Y);
			Shuttle24_Angel := LREAL_TO_REAL(gShuttleMon.Shuttle[24].Orientation.Angle1);
			Shuttle24_X := LREAL_TO_REAL(gShuttleMon.Shuttle[24].Position.X);
			Shuttle24_Y := LREAL_TO_REAL(gShuttleMon.Shuttle[24].Position.Y);
			Shuttle25_Angel := LREAL_TO_REAL(gShuttleMon.Shuttle[25].Orientation.Angle1);
			Shuttle25_X := LREAL_TO_REAL(gShuttleMon.Shuttle[25].Position.X);
			Shuttle25_Y := LREAL_TO_REAL(gShuttleMon.Shuttle[25].Position.Y);
			Shuttle26_Angel := LREAL_TO_REAL(gShuttleMon.Shuttle[26].Orientation.Angle1);
			Shuttle26_X := LREAL_TO_REAL(gShuttleMon.Shuttle[26].Position.X);
			Shuttle26_Y := LREAL_TO_REAL(gShuttleMon.Shuttle[26].Position.Y);
			Shuttle27_Angel := LREAL_TO_REAL(gShuttleMon.Shuttle[27].Orientation.Angle1);
			Shuttle27_X := LREAL_TO_REAL(gShuttleMon.Shuttle[27].Position.X);
			Shuttle27_Y := LREAL_TO_REAL(gShuttleMon.Shuttle[27].Position.Y);
			Shuttle28_Angel := LREAL_TO_REAL(gShuttleMon.Shuttle[28].Orientation.Angle1);
			Shuttle28_X := LREAL_TO_REAL(gShuttleMon.Shuttle[28].Position.X);
			Shuttle28_Y := LREAL_TO_REAL(gShuttleMon.Shuttle[28].Position.Y);
			Shuttle29_Angel := LREAL_TO_REAL(gShuttleMon.Shuttle[29].Orientation.Angle1);
			Shuttle29_X := LREAL_TO_REAL(gShuttleMon.Shuttle[29].Position.X);
			Shuttle29_Y := LREAL_TO_REAL(gShuttleMon.Shuttle[29].Position.Y);
			Shuttle30_Angel := LREAL_TO_REAL(gShuttleMon.Shuttle[30].Orientation.Angle1);
			Shuttle30_X := LREAL_TO_REAL(gShuttleMon.Shuttle[30].Position.X);
			Shuttle30_Y := LREAL_TO_REAL(gShuttleMon.Shuttle[30].Position.Y);
			Shuttle31_Angel := LREAL_TO_REAL(gShuttleMon.Shuttle[31].Orientation.Angle1);
			Shuttle31_X := LREAL_TO_REAL(gShuttleMon.Shuttle[31].Position.X);
			Shuttle31_Y := LREAL_TO_REAL(gShuttleMon.Shuttle[31].Position.Y);
			Shuttle32_Angel := LREAL_TO_REAL(gShuttleMon.Shuttle[32].Orientation.Angle1);
			Shuttle32_X := LREAL_TO_REAL(gShuttleMon.Shuttle[32].Position.X);
			Shuttle32_Y := LREAL_TO_REAL(gShuttleMon.Shuttle[32].Position.X);
			Shuttle33_Angel := LREAL_TO_REAL(gShuttleMon.Shuttle[33].Orientation.Angle1);
			Shuttle33_X := LREAL_TO_REAL(gShuttleMon.Shuttle[33].Position.X);
			Shuttle33_Y := LREAL_TO_REAL(gShuttleMon.Shuttle[33].Position.Y);
			Shuttle34_Angel := LREAL_TO_REAL(gShuttleMon.Shuttle[34].Orientation.Angle1);
			Shuttle34_X := LREAL_TO_REAL(gShuttleMon.Shuttle[34].Position.X);
			Shuttle34_Y := LREAL_TO_REAL(gShuttleMon.Shuttle[34].Position.Y);
			Shuttle35_Angel := LREAL_TO_REAL(gShuttleMon.Shuttle[35].Orientation.Angle1);
			Shuttle35_X := LREAL_TO_REAL(gShuttleMon.Shuttle[35].Position.X);
			Shuttle35_Y := LREAL_TO_REAL(gShuttleMon.Shuttle[35].Position.Y);
			Shuttle36_Angel := LREAL_TO_REAL(gShuttleMon.Shuttle[36].Orientation.Angle1);
			Shuttle36_X := LREAL_TO_REAL(gShuttleMon.Shuttle[36].Position.X);
			Shuttle36_Y := LREAL_TO_REAL(gShuttleMon.Shuttle[36].Position.Y);
			Shuttle37_Angel := LREAL_TO_REAL(gShuttleMon.Shuttle[37].Orientation.Angle1);
			Shuttle37_X := LREAL_TO_REAL(gShuttleMon.Shuttle[37].Position.X);
			Shuttle37_Y := LREAL_TO_REAL(gShuttleMon.Shuttle[37].Position.Y);
			Shuttle38_Angel := LREAL_TO_REAL(gShuttleMon.Shuttle[38].Orientation.Angle1);
			Shuttle38_X := LREAL_TO_REAL(gShuttleMon.Shuttle[38].Position.X);
			Shuttle38_Y := LREAL_TO_REAL(gShuttleMon.Shuttle[38].Position.Y);
			Shuttle39_Angel := LREAL_TO_REAL(gShuttleMon.Shuttle[39].Orientation.Angle1);
			Shuttle39_X := LREAL_TO_REAL(gShuttleMon.Shuttle[39].Position.X);
			Shuttle39_Y	:= LREAL_TO_REAL(gShuttleMon.Shuttle[39].Position.Y);
			Shuttle40_Angel := LREAL_TO_REAL(gShuttleMon.Shuttle[40].Orientation.Angle1);
			Shuttle40_X := LREAL_TO_REAL(gShuttleMon.Shuttle[40].Position.X);
			Shuttle40_Y := LREAL_TO_REAL(gShuttleMon.Shuttle[40].Position.Y);
			Shuttle41_Angel := LREAL_TO_REAL(gShuttleMon.Shuttle[41].Orientation.Angle1);
			Shuttle41_X := LREAL_TO_REAL(gShuttleMon.Shuttle[41].Position.X);
			Shuttle41_Y := LREAL_TO_REAL(gShuttleMon.Shuttle[41].Position.Y);
			Shuttle42_Angel := LREAL_TO_REAL(gShuttleMon.Shuttle[42].Orientation.Angle1);
			Shuttle42_X := LREAL_TO_REAL(gShuttleMon.Shuttle[42].Position.X);
			Shuttle42_Y := LREAL_TO_REAL(gShuttleMon.Shuttle[42].Position.Y);
			Shuttle43_Angel := LREAL_TO_REAL(gShuttleMon.Shuttle[43].Orientation.Angle1);
			Shuttle43_X := LREAL_TO_REAL(gShuttleMon.Shuttle[43].Position.X);
			Shuttle43_Y := LREAL_TO_REAL(gShuttleMon.Shuttle[43].Position.Y);
			Shuttle44_X := LREAL_TO_REAL(gShuttleMon.Shuttle[44].Position.X);
			Shuttle44_Y := LREAL_TO_REAL(gShuttleMon.Shuttle[44].Position.Y);
			Shuttle44_Angel := LREAL_TO_REAL(gShuttleMon.Shuttle[44].Orientation.Angle1);

		ELSE
			brsmemset(ADR(Vis.Shuttle[i]), 0, SIZEOF(Vis.Shuttle[0]));  //If the selected shuttle is not available, it will be invisible in the Scene Viewer
		END_IF
	END_FOR

END_PROGRAM
```

- Visualisation Logical/mappView (not shown)

### Program Logical/Safety (IEC)

#### Variables.var
```iecst
VAR
	moduleOK : BOOL;
	safetyStarted : BOOL;
	resetNeeded : BOOL;
	resetSafety : BOOL;
	safetyOK : BOOL;
END_VAR
```

#### Main.st
```iecst
PROGRAM _INIT
	(* Insert code here *)

END_PROGRAM

PROGRAM _CYCLIC
	IF resetNeeded THEN
		Safety_Status := 'Reset Needed';
	ELSIF safetyOK THEN
		Safety_Status := 'Safety OK';
	END_IF

END_PROGRAM

PROGRAM _EXIT
	(* Insert code here *)

END_PROGRAM
```

### Program Logical/SequenceHandler (IEC)

#### Variables.var
```iecst
VAR
	brestart : BOOL;
	bootmode : USINT := 1;
END_VAR
```

#### Main.st
```iecst
PROGRAM _INIT
	(* Insert code here *)
	AddJob :=FALSE;
	NeedPartcell1Bool :=FALSE;
	NeedPartCell2Bool :=FALSE;
	EmptyFixtureCell1Bool :=FALSE;
	EmptyFixtureCell2Bool :=FALSE;
	MoveAssemblyBool :=FALSE;
	brestart := FALSE;
END_PROGRAM

PROGRAM _CYCLIC
	(* Insert code here *)
	IF NeedPartcell1Bool AND EDGEPOS(AddJob) THEN
		NeedPartCell1 := NeedPartCell1 + 1;
	END_IF
	IF NeedPartCell2Bool AND EDGEPOS(AddJob) THEN
		NeedPartCell2 := NeedPartCell2 + 1;
	END_IF
	IF EmptyFixtureCell1Bool AND EDGEPOS(AddJob) THEN
		EmptyFixtureCell1 := EmptyFixtureCell1 + 1;
	END_IF
	IF EmptyFixtureCell2Bool AND EDGEPOS(AddJob) THEN
		EmptyFixtureCell2 := EmptyFixtureCell2 + 1;
	END_IF
	IF MoveAssemblyBool AND EDGEPOS(AddJob) THEN
		MoveAssemblyPart := MoveAssemblyPart + 1;
	END_IF
	IF MoveSubAssemblyPartBool AND EDGEPOS(AddJob) THEN
		MoveSubAssemblyPart := MoveAssemblyPart + 1;
	END_IF

	SYSreset(brestart,bootmode);

	IF EDGEPOS(AddJob) THEN
		NeedPartcell1Bool := FALSE;
		NeedPartCell2Bool := FALSE;
		EmptyFixtureCell1Bool := FALSE;
		EmptyFixtureCell2Bool := FALSE;
		MoveAssemblyBool := FALSE;
		MoveSubAssemblyPartBool := FALSE;
	END_IF

	IF HMILoadOffTrack AND WaitingLoadOff THEN
		LoadOffTrack := TRUE;
	END_IF
	IF HMILoadOnTrack AND WaitingLoadOn THEN
		LoadOnTrack := TRUE;
	END_IF
	IF HMITaskCompleteCell1 AND WaitingCell1 THEN
		TaskCompleteCell1 := TRUE;
	END_IF
	IF HMITaskCompleteCell2 AND WaitingCell2 THEN
		TaskCompleteCell2 := TRUE;
	END_IF

END_PROGRAM

PROGRAM _EXIT
	(* Insert code here *)

END_PROGRAM
```

### Program Logical/PB1 (IEC)

#### Variables.var
```iecst
VAR
	CmdEnableProcess : BOOL;
	CommandGiven : BOOL;
	MC_BR_BarrierCommand_AcpTrak_0 : MC_BR_BarrierCommand_AcpTrak;
	MC_BR_RoutedMoveAbs_AcpTrak_0 : MC_BR_RoutedMoveAbs_AcpTrak;
	MC_BR_ShCopyUserData_AcpTrak_0 : MC_BR_ShCopyUserData_AcpTrak;
	MC_BR_TrgPointEnable_AcpTrak_0 : MC_BR_TrgPointEnable_AcpTrak;
	MC_BR_TrgPointGetInfo_AcpTrak_0 : MC_BR_TrgPointGetInfo_AcpTrak;
	TON_0 : TON;
	PickupTimer : TON;
	ShuttleAxis : McAxisType;
	Speed_PP_04 : {REDUND_UNREPLICABLE} REAL := 0.0;
	Step : Step_enum;
	SubStep : UDINT;
	TaskReady : BOOL;
	WaitingCommand : BOOL;
	HMI_Barrier_Open : BOOL;
	HMI_Barrier_Close : BOOL;
	ShuttleUserData : ShuttleUserData_typ;
END_VAR
```

#### Cyclic.st
```iecst
PROGRAM _CYCLIC
	CASE Step OF
		CHECK_TRIGGER:
(* When the process is enabled and the assembly is ready,
the process will be activated *)
			IF((CmdEnableProcess) AND (gTrakAsm.Status.Ready))THEN
				MC_BR_TrgPointEnable_AcpTrak_0.Enable := TRUE;
(* If a shuttle passes the triggerpoint then
get the axis reference *)
				IF((MC_BR_TrgPointEnable_AcpTrak_0.Valid) AND
					(MC_BR_TrgPointEnable_AcpTrak_0.EventCount > 0))THEN
					MC_BR_TrgPointGetInfo_AcpTrak_0.Execute := TRUE;
				END_IF
			ELSE (* Else the processpoint will be disabled *)
				MC_BR_TrgPointEnable_AcpTrak_0.Enable := FALSE;
			END_IF
(* If axis reference is available,
save it AND go TO the next step *)
			IF EDGEPOS(MC_BR_TrgPointGetInfo_AcpTrak_0.Done) THEN
(* Save axis reference in local variable for use
in step machine *)
				ShuttleAxis := MC_BR_TrgPointGetInfo_AcpTrak_0.TrgPointInfo.Axis;
				MC_BR_TrgPointGetInfo_AcpTrak_0.Execute := FALSE;
				Step := GET_USERDATA;
				END_IF

		GET_USERDATA:
			(* The userdata is copied on a local variable *)
			MC_BR_ShCopyUserData_AcpTrak_0.Axis := ADR(ShuttleAxis);
			MC_BR_ShCopyUserData_AcpTrak_0.Execute := TRUE;
			MC_BR_ShCopyUserData_AcpTrak_0.DataAddress := ADR(ShuttleUserData);
			MC_BR_ShCopyUserData_AcpTrak_0.DataSize := SIZEOF(ShuttleUserData);
			MC_BR_ShCopyUserData_AcpTrak_0.Mode := mcACPTRAK_USERDATA_GET;
					(* After copying go to the next step *)

			IF EDGEPOS(MC_BR_ShCopyUserData_AcpTrak_0.Done) THEN
				MC_BR_ShCopyUserData_AcpTrak_0.Execute := FALSE;
				Step := PROCESS;
					END_IF

		PROCESS:

					IF 	MoveAssemblyPart >= 1 AND NOT Track6_Occupied THEN
						Track6_Occupied := TRUE;
						ShuttleUserData.State := InProcess;
						ShuttleUserData.Task := MoveAssembly;
						MoveAssemblyPart := MoveAssemblyPart-1;
						MC_BR_RoutedMoveAbs_AcpTrak_0.Execute := FALSE;
						PickupTimer.IN := TRUE;
						PickupTimer.PT := T#2s;
						WaitingCommand := FALSE;
						CommandGiven := TRUE;
						Step := SET_USERDATA;
					ELSIF 	EmptyFixtureCell1 >= 1 THEN
						ShuttleUserData.State := InProcess;
						ShuttleUserData.Task := PartsFromCell1;
						EmptyFixtureCell1 := EmptyFixtureCell1-1;
						MC_BR_RoutedMoveAbs_AcpTrak_0.Execute := FALSE;
						WaitingCommand := FALSE;
						CommandGiven := TRUE;
						Step := SET_USERDATA;
					ELSIF 	EmptyFixtureCell2 >= 1 THEN
						ShuttleUserData.State := InProcess;
						ShuttleUserData.Task := PartsFromCell2;
						EmptyFixtureCell2 := EmptyFixtureCell2-1;
						MC_BR_RoutedMoveAbs_AcpTrak_0.Execute := FALSE;
						WaitingCommand := FALSE;
						CommandGiven := TRUE;
						Step := SET_USERDATA;
					ELSIF	NeedPartCell1 >= 1 AND NOT Track6_Occupied THEN
						Track6_Occupied := TRUE;
						ShuttleUserData.State := InProcess;
						ShuttleUserData.Task := PartsToCell1;
						NeedPartCell1 := NeedPartCell1-1;
						MC_BR_RoutedMoveAbs_AcpTrak_0.Execute := FALSE;
						WaitingCommand := FALSE;
						CommandGiven := TRUE;
						PickupTimer.IN := TRUE;
						PickupTimer.PT := T#2s;
						Step := SET_USERDATA;
					ELSIF 	NeedPartCell2 >= 1 AND NOT Track6_Occupied THEN
						Track6_Occupied := TRUE;
						ShuttleUserData.State := InProcess;
						ShuttleUserData.Task := PartsToCell2;
						NeedPartCell2 := NeedPartCell2-1;
						MC_BR_RoutedMoveAbs_AcpTrak_0.Execute := FALSE;
						WaitingCommand := FALSE;
						CommandGiven := TRUE;
						PickupTimer.IN := TRUE;
						PickupTimer.PT := T#2s;
			  			Step := SET_USERDATA;
					ELSIF 	MoveSubAssemblyPart >= 1 AND NOT Track6_Occupied THEN
						Track6_Occupied := TRUE;
						ShuttleUserData.State := InProcess;
						ShuttleUserData.Task := MoveSubAssembly;
						MoveSubAssemblyPart := MoveSubAssemblyPart-1;
						MC_BR_RoutedMoveAbs_AcpTrak_0.Execute := FALSE;
						PickupTimer.IN := TRUE;
						PickupTimer.PT := T#2s;
						WaitingCommand := FALSE;
						CommandGiven := TRUE;
						Step := SET_USERDATA;
					ELSE
						ShuttleUserData.State := InProcess;
						ShuttleUserData.Task := NoTask;
						MC_BR_RoutedMoveAbs_AcpTrak_0.Execute := FALSE;
						WaitingCommand := FALSE;
						CommandGiven := TRUE;
						Step := SET_USERDATA;
					END_IF

		SET_USERDATA:
			(* The modified userdata will be copied back on the shuttle *)
			MC_BR_ShCopyUserData_AcpTrak_0.Axis := ADR(ShuttleAxis);
			MC_BR_ShCopyUserData_AcpTrak_0.Execute := TRUE;
			MC_BR_ShCopyUserData_AcpTrak_0.DataAddress := ADR(ShuttleUserData);
			MC_BR_ShCopyUserData_AcpTrak_0.DataSize := SIZEOF(ShuttleUserData);
			MC_BR_ShCopyUserData_AcpTrak_0.Mode := mcACPTRAK_USERDATA_SET;

			(* After copying go to the first step and wait for new event *)
			IF EDGEPOS(MC_BR_ShCopyUserData_AcpTrak_0.Done) THEN
				MC_BR_ShCopyUserData_AcpTrak_0.Execute := FALSE;
				Step := CHECK_TRIGGER;
			END_IF
	END_CASE

	IF EmptyFixtureCell1+EmptyFixtureCell2 >= 1 AND NOT CommandGiven AND NOT PickupTimer.IN AND NOT TON_0.IN AND NOT WaitingCommand THEN
		TaskReady := TRUE;
		MC_BR_BarrierCommand_AcpTrak_0.Command := 2;
		MC_BR_BarrierCommand_AcpTrak_0.Execute := TRUE;
		WaitingCommand := TRUE;
		TON_0.IN := TRUE;
		TON_0.PT :=T#500ms;
	ELSIF NeedPartCell1+NeedPartCell2+MoveAssemblyPart+MoveSubAssemblyPart >= 1 AND NOT CommandGiven AND NOT Track6_Occupied AND NOT TON_0.IN AND NOT WaitingCommand THEN
		TaskReady := TRUE;
		MC_BR_BarrierCommand_AcpTrak_0.Command := 2;
		MC_BR_BarrierCommand_AcpTrak_0.Execute := TRUE;
		WaitingCommand := TRUE;
		TON_0.IN := TRUE;
		TON_0.PT :=T#500ms;
	ELSE
		TaskReady := FALSE;
		MC_BR_BarrierCommand_AcpTrak_0.Execute := FALSE;
		CommandGiven := FALSE;
	END_IF

	IF TON_0.Q THEN
		TON_0.IN := FALSE;
	END_IF

	IF PickupTimer.Q THEN
		PickupTimer.IN := FALSE;
	END_IF

	IF EDGEPOS(HMI_Barrier_Open) THEN
		MC_BR_BarrierCommand_AcpTrak_0.Command := 0;
		MC_BR_BarrierCommand_AcpTrak_0.Execute := TRUE;
	ELSIF EDGEPOS(HMI_Barrier_Close) THEN
		MC_BR_BarrierCommand_AcpTrak_0.Command := 1;
		MC_BR_BarrierCommand_AcpTrak_0.Execute := TRUE;
	END_IF

	(* Call all function blocks *)
	MC_BR_TrgPointEnable_AcpTrak_0();
	MC_BR_TrgPointGetInfo_AcpTrak_0();
	MC_BR_ShCopyUserData_AcpTrak_0();
	MC_BR_RoutedMoveAbs_AcpTrak_0();
	MC_BR_BarrierCommand_AcpTrak_0();
	PickupTimer();
	TON_0();

END_PROGRAM
PROGRAM _EXIT
END_PROGRAM
```

#### Init.st
```iecst
PROGRAM _INIT
(* Local variable to enable/disable the the process *)
	Speed_PP_04 := 2;
	CmdEnableProcess := TRUE;
	(* Processpointreference for Functionblocks *)
	MC_BR_TrgPointEnable_AcpTrak_0.ProcessPoint := ADR(PB1);
	MC_BR_TrgPointGetInfo_AcpTrak_0.ProcessPoint := ADR(PB1);
	MC_BR_BarrierCommand_AcpTrak_0.ProcessPoint := ADR(PB1);
	MC_BR_BarrierCommand_AcpTrak_0.Command := 1;
	MC_BR_BarrierCommand_AcpTrak_0.AdvancedParameters.TicketCount := 1;
	MC_BR_BarrierCommand_AcpTrak_0.Execute := TRUE;
	MC_BR_BarrierCommand_AcpTrak_0();
	SubStep := 0;

END_PROGRAM
```

### Program Logical/PP1 (IEC)
